LIN {X 0,Y 523.9,Z 252.85,A -85,B 0,C 180,E1 -4806.401,E2 -4806.401} C_VEL
LIN {X 0,Y 523.917,Z 252.846,A -85,B 0,C 180,E1 -4809.084,E2 -4809.084} C_VEL
LIN {X 0,Y 523.952,Z 252.837,A -85,B 0,C 180,E1 -4812.118,E2 -4812.118} C_VEL
LIN {X 0,Y 523.95,Z 252.839,A -85,B 0,C 180,E1 -4815.308,E2 -4815.308} C_VEL
LIN {X 0,Y 523.956,Z 252.84,A -85,B 0,C 180,E1 -4818.688,E2 -4818.688} C_VEL
LIN {X 0,Y 523.912,Z 252.849,A -85,B 0,C 180,E1 -4821.898,E2 -4821.898} C_VEL
LIN {X 0,Y 523.933,Z 252.83,A -85,B 0,C 180,E1 -4824.908,E2 -4824.908} C_VEL
LIN {X 0,Y 523.936,Z 252.838,A -85,B 0,C 180,E1 -4827.678,E2 -4827.678} C_VEL
LIN {X 0,Y 523.963,Z 252.839,A -85,B 0,C 180,E1 -4830.673,E2 -4830.673} C_VEL
LIN {X 0,Y 523.971,Z 252.84,A -85,B 0,C 180,E1 -4833.728,E2 -4833.728} C_VEL
LIN {X 0,Y 523.929,Z 252.844,A -85,B 0,C 180,E1 -4836.27,E2 -4836.27} C_VEL
LIN {X 0,Y 523.938,Z 252.84,A -85,B 0,C 180,E1 -4838.766,E2 -4838.766} C_VEL
LIN {X 0,Y 523.946,Z 252.842,A -85,B 0,C 180,E1 -4841.221,E2 -4841.221} C_VEL
LIN {X 0,Y 523.933,Z 252.845,A -85,B 0,C 180,E1 -4843.639,E2 -4843.639} C_VEL
LIN {X 0,Y 523.933,Z 252.847,A -85,B 0,C 180,E1 -4846.028,E2 -4846.028} C_VEL
LIN {X 0,Y 524.003,Z 252.831,A -85,B 0,C 180,E1 -4848.394,E2 -4848.394} C_VEL
LIN {X 0,Y 523.997,Z 252.838,A -85,B 0,C 180,E1 -4851.516,E2 -4851.516} C_VEL
LIN {X 0,Y 524.076,Z 252.822,A -85,B 0,C 180,E1 -4854.614,E2 -4854.614} C_VEL
LIN {X 0,Y 524.103,Z 252.827,A -85,B 0,C 180,E1 -4857.694,E2 -4857.694} C_VEL
LIN {X 0,Y 524.117,Z 252.819,A -85,B 0,C 180,E1 -4860.768,E2 -4860.768} C_VEL
LIN {X 0,Y 524.067,Z 252.823,A -85,B 0,C 180,E1 -4863.075,E2 -4863.075} C_VEL
LIN {X 0,Y 524.038,Z 252.829,A -85,B 0,C 180,E1 -4866.159,E2 -4866.159} C_VEL
LIN {X 0,Y 523.993,Z 252.837,A -85,B 0,C 180,E1 -4869.262,E2 -4869.262} C_VEL
LIN {X 0,Y 523.994,Z 252.837,A -85,B 0,C 180,E1 -4871.74,E2 -4871.74} C_VEL
LIN {X 0,Y 523.984,Z 252.838,A -85,B 0,C 180,E1 -4875.053,E2 -4875.053} C_VEL
LIN {X 0,Y 523.957,Z 252.839,A -85,B 0,C 180,E1 -4877.969,E2 -4877.969} C_VEL
LIN {X 0,Y 523.964,Z 252.836,A -85,B 0,C 180,E1 -4880.41,E2 -4880.41} C_VEL
LIN {X 0,Y 523.909,Z 252.849,A -85,B 0,C 180,E1 -4882.894,E2 -4882.894} C_VEL
LIN {X 0,Y 523.946,Z 252.84,A -85,B 0,C 180,E1 -4885.419,E2 -4885.419} C_VEL
LIN {X 0,Y 523.964,Z 252.838,A -85,B 0,C 180,E1 -4887.999,E2 -4887.999} C_VEL
LIN {X 0,Y 523.947,Z 252.845,A -85,B 0,C 180,E1 -4890.857,E2 -4890.857} C_VEL
LIN {X 0,Y 523.956,Z 252.827,A -85,B 0,C 180,E1 -4893.736,E2 -4893.736} C_VEL
LIN {X 0,Y 523.917,Z 252.844,A -85,B 0,C 180,E1 -4896.405,E2 -4896.405} C_VEL
LIN {X 0,Y 523.919,Z 252.845,A -85,B 0,C 180,E1 -4899.085,E2 -4899.085} C_VEL
LIN {X 0,Y 523.952,Z 252.831,A -85,B 0,C 180,E1 -4902.119,E2 -4902.119} C_VEL
LIN {X 0,Y 523.952,Z 252.841,A -85,B 0,C 180,E1 -4905.309,E2 -4905.309} C_VEL
LIN {X 0,Y 523.92,Z 252.841,A -85,B 0,C 180,E1 -4906.92,E2 -4906.92} C_VEL
LIN {X 0,Y 523.253,Z 252.921,A -85,B 0,C 180,E1 -4907.561,E2 -4907.561} C_VEL
LIN {X 0,Y 520.408,Z 253.282,A -85,B 0,C 180,E1 -4908.603,E2 -4908.603} C_VEL
LIN {X 0,Y 518.002,Z 253.587,A -85,B 0,C 180,E1 -4909.442,E2 -4909.442} C_VEL
LIN {X 0,Y 516.965,Z 253.716,A -85,B 0,C 180,E1 -4910.089,E2 -4910.089} C_VEL
LIN {X 0,Y 516.879,Z 253.725,A -85,B 0,C 180,E1 -4910.309,E2 -4910.309} C_VEL
LIN {X 0,Y 516.882,Z 253.721,A -85,B 0,C 180,E1 -4913.343,E2 -4913.343} C_VEL
LIN {X 0,Y 516.91,Z 253.719,A -85,B 0,C 180,E1 -4916.122,E2 -4916.122} C_VEL
LIN {X 0,Y 516.891,Z 253.723,A -85,B 0,C 180,E1 -4918.936,E2 -4918.936} C_VEL
LIN {X 0,Y 516.919,Z 253.712,A -85,B 0,C 180,E1 -4921.585,E2 -4921.585} C_VEL
LIN {X 0,Y 516.93,Z 253.717,A -85,B 0,C 180,E1 -4924.211,E2 -4924.211} C_VEL
LIN {X 0,Y 516.93,Z 253.837,A -85,B 0,C 180,E1 -4925.929,E2 -4925.929} C_VEL
LIN {X 0,Y 518.632,Z 262.689,A -85,B 0,C 180,E1 -4927.53,E2 -4927.53} C_VEL
LIN {X 0,Y 518.198,Z 277.695,A -85,B 0,C 180,E1 -4929.974,E2 -4929.974} C_VEL
LIN {X 0,Y 517.98,Z 286.774,A -85,B 0,C 180,E1 -4931.404,E2 -4931.404} C_VEL
LIN {X 0,Y 520.284,Z 298.799,A -85,B 0,C 180,E1 -4931.688,E2 -4931.688} C_VEL
LIN {X 0,Y 520.017,Z 379.819,A -85,B 0,C 180,E1 -4932.83,E2 -4932.83} C_VEL
LIN {X 0,Y 519.682,Z 424.477,A -85,B 0,C 180,E1 -4933.476,E2 -4933.476} C_VEL
LIN {X 0,Y 519.367,Z 439.105,A -85,B 0,C 180,E1 -4933.852,E2 -4933.852} C_VEL
LIN {X 0,Y 519.086,Z 453.266,A -85,B 0,C 180,E1 -4934.39,E2 -4934.39} C_VEL
LIN {X 0,Y 518.692,Z 466.922,A -85,B 0,C 180,E1 -4935.082,E2 -4935.082} C_VEL
LIN {X 0,Y 518.257,Z 479.18,A -85,B 0,C 180,E1 -4935.872,E2 -4935.872} C_VEL
LIN {X 0,Y 517.892,Z 490.403,A -85,B 0,C 180,E1 -4936.762,E2 -4936.762} C_VEL
LIN {X 0,Y 517.497,Z 501.263,A -85,B 0,C 180,E1 -4937.803,E2 -4937.803} C_VEL
LIN {X 0,Y 517.151,Z 511.76,A -85,B 0,C 180,E1 -4939.032,E2 -4939.032} C_VEL
LIN {X 0,Y 516.844,Z 520.123,A -85,B 0,C 180,E1 -4940.214,E2 -4940.214} C_VEL
LIN {X 0,Y 516.605,Z 528.11,A -85,B 0,C 180,E1 -4941.591,E2 -4941.591} C_VEL
LIN {X 0,Y 516.418,Z 534.54,A -85,B 0,C 180,E1 -4942.965,E2 -4942.965} C_VEL
LIN {X 0,Y 516.391,Z 540.243,A -85,B 0,C 180,E1 -4944.533,E2 -4944.533} C_VEL
LIN {X 0,Y 516.343,Z 544.391,A -85,B 0,C 180,E1 -4946.098,E2 -4946.098} C_VEL
LIN {X 0,Y 516.26,Z 547.108,A -85,B 0,C 180,E1 -4947.659,E2 -4947.659} C_VEL
LIN {X 0,Y 516.156,Z 548.474,A -85,B 0,C 180,E1 -4949.22,E2 -4949.22} C_VEL
LIN {X 0,Y 516.157,Z 548.517,A -85,B 0,C 180,E1 -4950.78,E2 -4950.78} C_VEL
LIN {X 0,Y 516.26,Z 547.233,A -85,B 0,C 180,E1 -4952.341,E2 -4952.341} C_VEL
LIN {X 0,Y 516.343,Z 544.592,A -85,B 0,C 180,E1 -4953.902,E2 -4953.902} C_VEL
LIN {X 0,Y 516.39,Z 540.527,A -85,B 0,C 180,E1 -4955.467,E2 -4955.467} C_VEL
LIN {X 0,Y 516.414,Z 534.911,A -85,B 0,C 180,E1 -4957.035,E2 -4957.035} C_VEL
LIN {X 0,Y 516.6,Z 528.569,A -85,B 0,C 180,E1 -4958.409,E2 -4958.409} C_VEL
LIN {X 0,Y 516.824,Z 520.683,A -85,B 0,C 180,E1 -4959.786,E2 -4959.786} C_VEL
LIN {X 0,Y 517.115,Z 512.434,A -85,B 0,C 180,E1 -4960.968,E2 -4960.968} C_VEL
LIN {X 0,Y 517.445,Z 502.412,A -85,B 0,C 180,E1 -4962.162,E2 -4962.162} C_VEL
LIN {X 0,Y 517.814,Z 491.436,A -85,B 0,C 180,E1 -4963.24,E2 -4963.24} C_VEL
LIN {X 0,Y 518.21,Z 480.425,A -85,B 0,C 180,E1 -4964.129,E2 -4964.129} C_VEL
LIN {X 0,Y 518.681,Z 468.481,A -85,B 0,C 180,E1 -4964.918,E2 -4964.918} C_VEL
LIN {X 0,Y 519.054,Z 455.296,A -85,B 0,C 180,E1 -4965.611,E2 -4965.611} C_VEL
LIN {X 0,Y 519.377,Z 441.413,A -85,B 0,C 180,E1 -4966.161,E2 -4966.161} C_VEL
LIN {X 0,Y 519.651,Z 427.406,A -85,B 0,C 180,E1 -4966.55,E2 -4966.55} C_VEL
LIN {X 0,Y 519.811,Z 409.431,A -85,B 0,C 180,E1 -4966.848,E2 -4966.848} C_VEL
LIN {X 0,Y 520.381,Z 299.087,A -85,B 0,C 180,E1 -4968.394,E2 -4968.394} C_VEL
LIN {X 0,Y 517.983,Z 286.806,A -85,B 0,C 180,E1 -4968.684,E2 -4968.684} C_VEL
LIN {X 0,Y 518.506,Z 269.351,A -85,B 0,C 180,E1 -4971.467,E2 -4971.467} C_VEL
LIN {X 0,Y 518.596,Z 262.055,A -85,B 0,C 180,E1 -4972.667,E2 -4972.667} C_VEL
LIN {X 0,Y 516.909,Z 253.814,A -85,B 0,C 180,E1 -4974.173,E2 -4974.173} C_VEL
LIN {X 0,Y 516.927,Z 253.719,A -85,B 0,C 180,E1 -4976.657,E2 -4976.657} C_VEL
LIN {X 0,Y 516.91,Z 253.719,A -85,B 0,C 180,E1 -4979.523,E2 -4979.523} C_VEL
LIN {X 0,Y 516.896,Z 253.72,A -85,B 0,C 180,E1 -4982.543,E2 -4982.543} C_VEL
LIN {X 0,Y 516.878,Z 253.725,A -85,B 0,C 180,E1 -4985.331,E2 -4985.331} C_VEL
LIN {X 0,Y 516.878,Z 253.722,A -85,B 0,C 180,E1 -4987.942,E2 -4987.942} C_VEL
LIN {X 0,Y 516.883,Z 253.722,A -85,B 0,C 180,E1 -4990.741,E2 -4990.741} C_VEL
LIN {X 0,Y 516.901,Z 253.712,A -85,B 0,C 180,E1 -4992.828,E2 -4992.828} C_VEL
LIN {X 0,Y 516.919,Z 253.719,A -85,B 0,C 180,E1 -4995.009,E2 -4995.009} C_VEL
LIN {X 0,Y 516.917,Z 253.706,A -85,B 0,C 180,E1 -4998.397,E2 -4998.397} C_VEL
LIN {X 0,Y 516.881,Z 253.727,A -85,B 0,C 180,E1 -5001.284,E2 -5001.284} C_VEL
LIN {X 0,Y 516.885,Z 253.718,A -85,B 0,C 180,E1 -5004.221,E2 -5004.221} C_VEL
LIN {X 0,Y 516.891,Z 253.711,A -85,B 0,C 180,E1 -5007.053,E2 -5007.053} C_VEL
LIN {X 0,Y 516.895,Z 253.719,A -85,B 0,C 180,E1 -5009.796,E2 -5009.796} C_VEL
LIN {X 0,Y 516.921,Z 253.717,A -85,B 0,C 180,E1 -5012.467,E2 -5012.467} C_VEL
LIN {X 0,Y 516.903,Z 253.724,A -85,B 0,C 180,E1 -5015.071,E2 -5015.071} C_VEL
LIN {X 0,Y 516.861,Z 253.723,A -85,B 0,C 180,E1 -5017.621,E2 -5017.621} C_VEL
LIN {X 0,Y 516.924,Z 253.712,A -85,B 0,C 180,E1 -5020.129,E2 -5020.129} C_VEL
LIN {X 0,Y 516.923,Z 253.72,A -85,B 0,C 180,E1 -5022.596,E2 -5022.596} C_VEL
LIN {X 0,Y 516.933,Z 253.716,A -85,B 0,C 180,E1 -5025.03,E2 -5025.03} C_VEL
LIN {X 0,Y 516.956,Z 253.713,A -85,B 0,C 180,E1 -5028.233,E2 -5028.233} C_VEL
LIN {X 0,Y 516.961,Z 253.706,A -85,B 0,C 180,E1 -5031.399,E2 -5031.399} C_VEL
LIN {X 0,Y 517.002,Z 253.705,A -85,B 0,C 180,E1 -5033.757,E2 -5033.757} C_VEL
LIN {X 0,Y 517.008,Z 253.703,A -85,B 0,C 180,E1 -5036.883,E2 -5036.883} C_VEL
LIN {X 0,Y 517.075,Z 253.697,A -85,B 0,C 180,E1 -5040,E2 -5040} C_VEL
LIN {X 0,Y 517.008,Z 253.701,A -85,B 0,C 180,E1 -5043.117,E2 -5043.117} C_VEL
LIN {X 0,Y 517.001,Z 253.71,A -85,B 0,C 180,E1 -5046.243,E2 -5046.243} C_VEL
LIN {X 0,Y 516.948,Z 253.709,A -85,B 0,C 180,E1 -5049.389,E2 -5049.389} C_VEL
LIN {X 0,Y 516.942,Z 253.712,A -85,B 0,C 180,E1 -5051.807,E2 -5051.807} C_VEL
LIN {X 0,Y 516.935,Z 253.712,A -85,B 0,C 180,E1 -5055.147,E2 -5055.147} C_VEL
LIN {X 0,Y 516.917,Z 253.723,A -85,B 0,C 180,E1 -5058.222,E2 -5058.222} C_VEL
LIN {X 0,Y 516.903,Z 253.717,A -85,B 0,C 180,E1 -5060.702,E2 -5060.702} C_VEL
LIN {X 0,Y 516.903,Z 253.725,A -85,B 0,C 180,E1 -5064.072,E2 -5064.072} C_VEL
LIN {X 0,Y 516.918,Z 253.714,A -85,B 0,C 180,E1 -5066.658,E2 -5066.658} C_VEL
LIN {X 0,Y 516.917,Z 253.718,A -85,B 0,C 180,E1 -5069.527,E2 -5069.527} C_VEL
LIN {X 0,Y 516.893,Z 253.713,A -85,B 0,C 180,E1 -5072.545,E2 -5072.545} C_VEL
LIN {X 0,Y 516.876,Z 253.71,A -85,B 0,C 180,E1 -5075.333,E2 -5075.333} C_VEL
LIN {X 0,Y 516.876,Z 253.729,A -85,B 0,C 180,E1 -5077.944,E2 -5077.944} C_VEL
LIN {X 0,Y 516.88,Z 253.718,A -85,B 0,C 180,E1 -5080.742,E2 -5080.742} C_VEL
LIN {X 0,Y 516.878,Z 253.721,A -85,B 0,C 180,E1 -5082.832,E2 -5082.832} C_VEL
LIN {X 0,Y 516.918,Z 253.716,A -85,B 0,C 180,E1 -5085.011,E2 -5085.011} C_VEL
LIN {X 0,Y 516.919,Z 253.71,A -85,B 0,C 180,E1 -5088.398,E2 -5088.398} C_VEL
LIN {X 0,Y 516.882,Z 253.726,A -85,B 0,C 180,E1 -5091.285,E2 -5091.285} C_VEL
LIN {X 0,Y 516.868,Z 253.724,A -85,B 0,C 180,E1 -5094.22,E2 -5094.22} C_VEL
LIN {X 0,Y 516.894,Z 253.719,A -85,B 0,C 180,E1 -5097.054,E2 -5097.054} C_VEL
LIN {X 0,Y 516.891,Z 253.709,A -85,B 0,C 180,E1 -5099.797,E2 -5099.797} C_VEL
LIN {X 0,Y 516.927,Z 253.719,A -85,B 0,C 180,E1 -5102.468,E2 -5102.468} C_VEL
LIN {X 0,Y 516.955,Z 253.758,A -85,B 0,C 180,E1 -5104.752,E2 -5104.752} C_VEL
LIN {X 0,Y 517.3,Z 255.393,A -85,B 0,C 180,E1 -5105.093,E2 -5105.093} C_VEL
LIN {X 0,Y 518.896,Z 263.487,A -85,B 0,C 180,E1 -5106.45,E2 -5106.45} C_VEL
LIN {X 0,Y 518.406,Z 279.65,A -85,B 0,C 180,E1 -5108.946,E2 -5108.946} C_VEL
LIN {X 0,Y 518.002,Z 295.678,A -85,B 0,C 180,E1 -5111.358,E2 -5111.358} C_VEL
LIN {X 0,Y 520.437,Z 309.426,A -85,B 0,C 180,E1 -5111.668,E2 -5111.668} C_VEL
LIN {X 0,Y 519.66,Z 433.577,A -85,B 0,C 180,E1 -5113.425,E2 -5113.425} C_VEL
LIN {X 0,Y 519.376,Z 447.528,A -85,B 0,C 180,E1 -5113.777,E2 -5113.777} C_VEL
LIN {X 0,Y 519.085,Z 461.402,A -85,B 0,C 180,E1 -5114.289,E2 -5114.289} C_VEL
LIN {X 0,Y 518.753,Z 473.578,A -85,B 0,C 180,E1 -5114.883,E2 -5114.883} C_VEL
LIN {X 0,Y 518.282,Z 486.388,A -85,B 0,C 180,E1 -5115.672,E2 -5115.672} C_VEL
LIN {X 0,Y 517.89,Z 498.036,A -85,B 0,C 180,E1 -5116.562,E2 -5116.562} C_VEL
LIN {X 0,Y 517.493,Z 508.974,A -85,B 0,C 180,E1 -5117.577,E2 -5117.577} C_VEL
LIN {X 0,Y 517.235,Z 518.468,A -85,B 0,C 180,E1 -5118.638,E2 -5118.638} C_VEL
LIN {X 0,Y 516.849,Z 527.332,A -85,B 0,C 180,E1 -5119.819,E2 -5119.819} C_VEL
LIN {X 0,Y 516.683,Z 534.708,A -85,B 0,C 180,E1 -5121.001,E2 -5121.001} C_VEL
LIN {X 0,Y 516.495,Z 540.857,A -85,B 0,C 180,E1 -5122.18,E2 -5122.18} C_VEL
LIN {X 0,Y 516.382,Z 547.387,A -85,B 0,C 180,E1 -5123.749,E2 -5123.749} C_VEL
LIN {X 0,Y 516.305,Z 551.207,A -85,B 0,C 180,E1 -5124.924,E2 -5124.924} C_VEL
LIN {X 0,Y 516.324,Z 554.15,A -85,B 0,C 180,E1 -5126.098,E2 -5126.098} C_VEL
LIN {X 0,Y 516.259,Z 556.844,A -85,B 0,C 180,E1 -5127.659,E2 -5127.659} C_VEL
LIN {X 0,Y 516.157,Z 558.178,A -85,B 0,C 180,E1 -5129.22,E2 -5129.22} C_VEL
LIN {X 0,Y 516.157,Z 558.178,A -85,B 0,C 180,E1 -5130.78,E2 -5130.78} C_VEL
LIN {X 0,Y 516.26,Z 556.847,A -85,B 0,C 180,E1 -5132.341,E2 -5132.341} C_VEL
LIN {X 0,Y 516.324,Z 554.154,A -85,B 0,C 180,E1 -5133.902,E2 -5133.902} C_VEL
LIN {X 0,Y 516.382,Z 550.026,A -85,B 0,C 180,E1 -5135.467,E2 -5135.467} C_VEL
LIN {X 0,Y 516.402,Z 544.337,A -85,B 0,C 180,E1 -5137.035,E2 -5137.035} C_VEL
LIN {X 0,Y 516.582,Z 537.923,A -85,B 0,C 180,E1 -5138.41,E2 -5138.41} C_VEL
LIN {X 0,Y 516.805,Z 529.954,A -85,B 0,C 180,E1 -5139.787,E2 -5139.787} C_VEL
LIN {X 0,Y 517.101,Z 521.618,A -85,B 0,C 180,E1 -5140.969,E2 -5140.969} C_VEL
LIN {X 0,Y 517.456,Z 511.182,A -85,B 0,C 180,E1 -5142.197,E2 -5142.197} C_VEL
LIN {X 0,Y 517.824,Z 500.382,A -85,B 0,C 180,E1 -5143.24,E2 -5143.24} C_VEL
LIN {X 0,Y 518.245,Z 487.817,A -85,B 0,C 180,E1 -5144.229,E2 -5144.229} C_VEL
LIN {X 0,Y 518.7,Z 475.343,A -85,B 0,C 180,E1 -5145.018,E2 -5145.018} C_VEL
LIN {X 0,Y 519.077,Z 462.519,A -85,B 0,C 180,E1 -5145.661,E2 -5145.661} C_VEL
LIN {X 0,Y 519.367,Z 448.602,A -85,B 0,C 180,E1 -5146.188,E2 -5146.188} C_VEL
LIN {X 0,Y 519.65,Z 434.709,A -85,B 0,C 180,E1 -5146.55,E2 -5146.55} C_VEL
LIN {X 0,Y 519.847,Z 408.415,A -85,B 0,C 180,E1 -5146.948,E2 -5146.948} C_VEL
LIN {X 0,Y 520.279,Z 308.185,A -85,B 0,C 180,E1 -5148.355,E2 -5148.355} C_VEL
LIN {X 0,Y 517.994,Z 295.748,A -85,B 0,C 180,E1 -5148.638,E2 -5148.638} C_VEL
LIN {X 0,Y 518.507,Z 276.952,A -85,B 0,C 180,E1 -5151.467,E2 -5151.467} C_VEL
LIN {X 0,Y 518.89,Z 263.487,A -85,B 0,C 180,E1 -5153.55,E2 -5153.55} C_VEL
LIN {X 0,Y 517.034,Z 254.105,A -85,B 0,C 180,E1 -5155.136,E2 -5155.136} C_VEL
LIN {X 0,Y 516.954,Z 253.708,A -85,B 0,C 180,E1 -5155.356,E2 -5155.356} C_VEL
LIN {X 0,Y 516.918,Z 253.718,A -85,B 0,C 180,E1 -5158.415,E2 -5158.415} C_VEL
LIN {X 0,Y 516.888,Z 253.723,A -85,B 0,C 180,E1 -5161.109,E2 -5161.109} C_VEL
LIN {X 0,Y 516.906,Z 253.716,A -85,B 0,C 180,E1 -5163.966,E2 -5163.966} C_VEL
LIN {X 0,Y 516.873,Z 253.722,A -85,B 0,C 180,E1 -5166.745,E2 -5166.745} C_VEL
LIN {X 0,Y 516.878,Z 253.722,A -85,B 0,C 180,E1 -5169.721,E2 -5169.721} C_VEL
LIN {X 0,Y 516.902,Z 253.721,A -85,B 0,C 180,E1 -5172.76,E2 -5172.76} C_VEL
LIN {X 0,Y 516.918,Z 253.716,A -85,B 0,C 180,E1 -5175.009,E2 -5175.009} C_VEL
LIN {X 0,Y 516.912,Z 253.721,A -85,B 0,C 180,E1 -5178.398,E2 -5178.398} C_VEL
LIN {X 0,Y 516.878,Z 253.721,A -85,B 0,C 180,E1 -5181.284,E2 -5181.284} C_VEL
LIN {X 0,Y 516.885,Z 253.715,A -85,B 0,C 180,E1 -5184.221,E2 -5184.221} C_VEL
LIN {X 0,Y 516.891,Z 253.712,A -85,B 0,C 180,E1 -5187.053,E2 -5187.053} C_VEL
LIN {X 0,Y 516.895,Z 253.723,A -85,B 0,C 180,E1 -5189.797,E2 -5189.797} C_VEL
LIN {X 0,Y 516.923,Z 253.715,A -85,B 0,C 180,E1 -5192.467,E2 -5192.467} C_VEL
LIN {X 0,Y 516.904,Z 253.718,A -85,B 0,C 180,E1 -5195.072,E2 -5195.072} C_VEL
LIN {X 0,Y 516.878,Z 253.721,A -85,B 0,C 180,E1 -5198.462,E2 -5198.462} C_VEL
LIN {X 0,Y 516.897,Z 253.719,A -85,B 0,C 180,E1 -5200.955,E2 -5200.955} C_VEL
LIN {X 0,Y 516.909,Z 253.717,A -85,B 0,C 180,E1 -5203.41,E2 -5203.41} C_VEL
LIN {X 0,Y 516.888,Z 253.728,A -85,B 0,C 180,E1 -5205.833,E2 -5205.833} C_VEL
LIN {X 0,Y 516.957,Z 253.71,A -85,B 0,C 180,E1 -5208.234,E2 -5208.234} C_VEL
LIN {X 0,Y 516.962,Z 253.712,A -85,B 0,C 180,E1 -5211.4,E2 -5211.4} C_VEL
LIN {X 0,Y 517.002,Z 253.71,A -85,B 0,C 180,E1 -5213.757,E2 -5213.757} C_VEL
LIN {X 0,Y 517.076,Z 253.703,A -85,B 0,C 180,E1 -5217.663,E2 -5217.663} C_VEL
LIN {X 0,Y 517.087,Z 253.694,A -85,B 0,C 180,E1 -5220.779,E2 -5220.779} C_VEL
LIN {X 0,Y 517.008,Z 253.702,A -85,B 0,C 180,E1 -5223.117,E2 -5223.117} C_VEL
LIN {X 0,Y 517.002,Z 253.705,A -85,B 0,C 180,E1 -5226.243,E2 -5226.243} C_VEL
LIN {X 0,Y 516.947,Z 253.715,A -85,B 0,C 180,E1 -5229.389,E2 -5229.389} C_VEL
LIN {X 0,Y 516.944,Z 253.715,A -85,B 0,C 180,E1 -5231.808,E2 -5231.808} C_VEL
LIN {X 0,Y 516.936,Z 253.716,A -85,B 0,C 180,E1 -5235.147,E2 -5235.147} C_VEL
LIN {X 0,Y 516.918,Z 253.716,A -85,B 0,C 180,E1 -5238.223,E2 -5238.223} C_VEL
LIN {X 0,Y 516.905,Z 253.717,A -85,B 0,C 180,E1 -5240.702,E2 -5240.702} C_VEL
LIN {X 0,Y 516.904,Z 253.718,A -85,B 0,C 180,E1 -5244.072,E2 -5244.072} C_VEL
LIN {X 0,Y 516.92,Z 253.715,A -85,B 0,C 180,E1 -5246.658,E2 -5246.658} C_VEL
LIN {X 0,Y 516.919,Z 253.717,A -85,B 0,C 180,E1 -5249.527,E2 -5249.527} C_VEL
LIN {X 0,Y 516.895,Z 253.715,A -85,B 0,C 180,E1 -5252.545,E2 -5252.545} C_VEL
LIN {X 0,Y 516.878,Z 253.72,A -85,B 0,C 180,E1 -5255.333,E2 -5255.333} C_VEL
LIN {X 0,Y 516.877,Z 253.722,A -85,B 0,C 180,E1 -5257.944,E2 -5257.944} C_VEL
LIN {X 0,Y 516.899,Z 253.715,A -85,B 0,C 180,E1 -5260.74,E2 -5260.74} C_VEL
LIN {X 0,Y 516.879,Z 253.72,A -85,B 0,C 180,E1 -5263.904,E2 -5263.904} C_VEL
LIN {X 0,Y 516.879,Z 253.722,A -85,B 0,C 180,E1 -5266.108,E2 -5266.108} C_VEL
LIN {X 0,Y 516.915,Z 253.714,A -85,B 0,C 180,E1 -5268.399,E2 -5268.399} C_VEL
LIN {X 0,Y 516.879,Z 253.725,A -85,B 0,C 180,E1 -5270.309,E2 -5270.309} C_VEL
LIN {X 0,Y 516.209,Z 253.807,A -85,B 0,C 180,E1 -5270.959,E2 -5270.959} C_VEL
LIN {X 0,Y 513.364,Z 254.159,A -85,B 0,C 180,E1 -5272.015,E2 -5272.015} C_VEL
LIN {X 0,Y 510.956,Z 254.463,A -85,B 0,C 180,E1 -5272.865,E2 -5272.865} C_VEL
LIN {X 0,Y 509.916,Z 254.589,A -85,B 0,C 180,E1 -5273.521,E2 -5273.521} C_VEL
LIN {X 0,Y 509.828,Z 254.6,A -85,B 0,C 180,E1 -5273.744,E2 -5273.744} C_VEL
LIN {X 0,Y 509.86,Z 254.6,A -85,B 0,C 180,E1 -5276.54,E2 -5276.54} C_VEL
LIN {X 0,Y 509.845,Z 254.599,A -85,B 0,C 180,E1 -5279.335,E2 -5279.335} C_VEL
LIN {X 0,Y 509.894,Z 254.585,A -85,B 0,C 180,E1 -5282.055,E2 -5282.055} C_VEL
LIN {X 0,Y 509.841,Z 254.593,A -85,B 0,C 180,E1 -5284.703,E2 -5284.703} C_VEL
LIN {X 0,Y 509.875,Z 254.64,A -85,B 0,C 180,E1 -5285.683,E2 -5285.683} C_VEL
LIN {X 0,Y 510.429,Z 257.459,A -85,B 0,C 180,E1 -5286.251,E2 -5286.251} C_VEL
LIN {X 0,Y 511.783,Z 265.056,A -85,B 0,C 180,E1 -5287.6,E2 -5287.6} C_VEL
LIN {X 0,Y 511.126,Z 282.841,A -85,B 0,C 180,E1 -5290.523,E2 -5290.523} C_VEL
LIN {X 0,Y 511.067,Z 286.884,A -85,B 0,C 180,E1 -5291.146,E2 -5291.146} C_VEL
LIN {X 0,Y 513.675,Z 300.421,A -85,B 0,C 180,E1 -5291.466,E2 -5291.466} C_VEL
LIN {X 0,Y 512.899,Z 423.387,A -85,B 0,C 180,E1 -5293.226,E2 -5293.226} C_VEL
LIN {X 0,Y 512.57,Z 438.113,A -85,B 0,C 180,E1 -5293.596,E2 -5293.596} C_VEL
LIN {X 0,Y 512.284,Z 452.218,A -85,B 0,C 180,E1 -5294.126,E2 -5294.126} C_VEL
LIN {X 0,Y 511.912,Z 465.234,A -85,B 0,C 180,E1 -5294.778,E2 -5294.778} C_VEL
LIN {X 0,Y 511.412,Z 477.832,A -85,B 0,C 180,E1 -5295.577,E2 -5295.577} C_VEL
LIN {X 0,Y 510.999,Z 489.305,A -85,B 0,C 180,E1 -5296.479,E2 -5296.479} C_VEL
LIN {X 0,Y 510.55,Z 499.789,A -85,B 0,C 180,E1 -5297.474,E2 -5297.474} C_VEL
LIN {X 0,Y 510.208,Z 510.284,A -85,B 0,C 180,E1 -5298.68,E2 -5298.68} C_VEL
LIN {X 0,Y 509.836,Z 518.905,A -85,B 0,C 180,E1 -5299.878,E2 -5299.878} C_VEL
LIN {X 0,Y 509.602,Z 527.17,A -85,B 0,C 180,E1 -5301.275,E2 -5301.275} C_VEL
LIN {X 0,Y 509.413,Z 532.927,A -85,B 0,C 180,E1 -5302.469,E2 -5302.469} C_VEL
LIN {X 0,Y 509.308,Z 537.665,A -85,B 0,C 180,E1 -5303.662,E2 -5303.662} C_VEL
LIN {X 0,Y 509.239,Z 541.51,A -85,B 0,C 180,E1 -5304.853,E2 -5304.853} C_VEL
LIN {X 0,Y 509.251,Z 544.459,A -85,B 0,C 180,E1 -5306.043,E2 -5306.043} C_VEL
LIN {X 0,Y 509.189,Z 547.175,A -85,B 0,C 180,E1 -5307.627,E2 -5307.627} C_VEL
LIN {X 0,Y 509.07,Z 548.541,A -85,B 0,C 180,E1 -5309.209,E2 -5309.209} C_VEL
LIN {X 0,Y 509.071,Z 548.584,A -85,B 0,C 180,E1 -5310.791,E2 -5310.791} C_VEL
LIN {X 0,Y 509.188,Z 547.299,A -85,B 0,C 180,E1 -5312.373,E2 -5312.373} C_VEL
LIN {X 0,Y 509.251,Z 544.657,A -85,B 0,C 180,E1 -5313.957,E2 -5313.957} C_VEL
LIN {X 0,Y 509.327,Z 540.592,A -85,B 0,C 180,E1 -5315.543,E2 -5315.543} C_VEL
LIN {X 0,Y 509.361,Z 534.975,A -85,B 0,C 180,E1 -5317.133,E2 -5317.133} C_VEL
LIN {X 0,Y 509.557,Z 528.633,A -85,B 0,C 180,E1 -5318.526,E2 -5318.526} C_VEL
LIN {X 0,Y 509.783,Z 520.746,A -85,B 0,C 180,E1 -5319.923,E2 -5319.923} C_VEL
LIN {X 0,Y 510.114,Z 512.496,A -85,B 0,C 180,E1 -5321.121,E2 -5321.121} C_VEL
LIN {X 0,Y 510.455,Z 502.828,A -85,B 0,C 180,E1 -5322.291,E2 -5322.291} C_VEL
LIN {X 0,Y 510.898,Z 491.496,A -85,B 0,C 180,E1 -5323.422,E2 -5323.422} C_VEL
LIN {X 0,Y 511.314,Z 480.484,A -85,B 0,C 180,E1 -5324.324,E2 -5324.324} C_VEL
LIN {X 0,Y 511.819,Z 468.537,A -85,B 0,C 180,E1 -5325.123,E2 -5325.123} C_VEL
LIN {X 0,Y 512.219,Z 455.348,A -85,B 0,C 180,E1 -5325.825,E2 -5325.825} C_VEL
LIN {X 0,Y 512.557,Z 441.104,A -85,B 0,C 180,E1 -5326.394,E2 -5326.394} C_VEL
LIN {X 0,Y 512.841,Z 427.444,A -85,B 0,C 180,E1 -5326.776,E2 -5326.776} C_VEL
LIN {X 0,Y 513.01,Z 407.664,A -85,B 0,C 180,E1 -5327.104,E2 -5327.104} C_VEL
LIN {X 0,Y 513.652,Z 299.991,A -85,B 0,C 180,E1 -5328.631,E2 -5328.631} C_VEL
LIN {X 0,Y 511.089,Z 287.082,A -85,B 0,C 180,E1 -5328.933,E2 -5328.933} C_VEL
LIN {X 0,Y 511.095,Z 284.659,A -85,B 0,C 180,E1 -5329.27,E2 -5329.27} C_VEL
LIN {X 0,Y 511.794,Z 265.599,A -85,B 0,C 180,E1 -5332.399,E2 -5332.399} C_VEL
LIN {X 0,Y 510.847,Z 259.261,A -85,B 0,C 180,E1 -5333.513,E2 -5333.513} C_VEL
LIN {X 0,Y 509.878,Z 254.731,A -85,B 0,C 180,E1 -5334.371,E2 -5334.371} C_VEL
LIN {X 0,Y 509.886,Z 254.596,A -85,B 0,C 180,E1 -5337.055,E2 -5337.055} C_VEL
LIN {X 0,Y 509.856,Z 254.602,A -85,B 0,C 180,E1 -5339.75,E2 -5339.75} C_VEL
LIN {X 0,Y 509.873,Z 254.595,A -85,B 0,C 180,E1 -5342.774,E2 -5342.774} C_VEL
LIN {X 0,Y 509.837,Z 254.606,A -85,B 0,C 180,E1 -5345.58,E2 -5345.58} C_VEL
LIN {X 0,Y 509.847,Z 254.595,A -85,B 0,C 180,E1 -5348.337,E2 -5348.337} C_VEL
LIN {X 0,Y 509.855,Z 254.598,A -85,B 0,C 180,E1 -5351.424,E2 -5351.424} C_VEL
LIN {X 0,Y 509.853,Z 254.596,A -85,B 0,C 180,E1 -5354.667,E2 -5354.667} C_VEL
LIN {X 0,Y 509.856,Z 254.585,A -85,B 0,C 180,E1 -5358.102,E2 -5358.102} C_VEL
LIN {X 0,Y 509.854,Z 254.594,A -85,B 0,C 180,E1 -5360.648,E2 -5360.648} C_VEL
LIN {X 0,Y 509.83,Z 254.6,A -85,B 0,C 180,E1 -5363.647,E2 -5363.647} C_VEL
LIN {X 0,Y 509.856,Z 254.584,A -85,B 0,C 180,E1 -5366.539,E2 -5366.539} C_VEL
LIN {X 0,Y 509.844,Z 254.603,A -85,B 0,C 180,E1 -5369.334,E2 -5369.334} C_VEL
LIN {X 0,Y 509.887,Z 254.592,A -85,B 0,C 180,E1 -5372.054,E2 -5372.054} C_VEL
LIN {X 0,Y 509.869,Z 254.594,A -85,B 0,C 180,E1 -5374.703,E2 -5374.703} C_VEL
LIN {X 0,Y 509.819,Z 254.601,A -85,B 0,C 180,E1 -5377.457,E2 -5377.457} C_VEL
LIN {X 0,Y 509.908,Z 254.586,A -85,B 0,C 180,E1 -5379.844,E2 -5379.844} C_VEL
LIN {X 0,Y 509.879,Z 254.595,A -85,B 0,C 180,E1 -5383.174,E2 -5383.174} C_VEL
LIN {X 0,Y 509.855,Z 254.592,A -85,B 0,C 180,E1 -5385.634,E2 -5385.634} C_VEL
LIN {X 0,Y 509.909,Z 254.594,A -85,B 0,C 180,E1 -5388.874,E2 -5388.874} C_VEL
LIN {X 0,Y 509.942,Z 254.581,A -85,B 0,C 180,E1 -5392.078,E2 -5392.078} C_VEL
LIN {X 0,Y 509.984,Z 254.586,A -85,B 0,C 180,E1 -5394.464,E2 -5394.464} C_VEL
LIN {X 0,Y 510.046,Z 254.565,A -85,B 0,C 180,E1 -5397.631,E2 -5397.631} C_VEL
LIN {X 0,Y 510.057,Z 254.575,A -85,B 0,C 180,E1 -5400.789,E2 -5400.789} C_VEL
LIN {X 0,Y 509.95,Z 254.58,A -85,B 0,C 180,E1 -5403.16,E2 -5403.16} C_VEL
LIN {X 0,Y 509.97,Z 254.587,A -85,B 0,C 180,E1 -5406.33,E2 -5406.33} C_VEL
LIN {X 0,Y 509.909,Z 254.589,A -85,B 0,C 180,E1 -5408.72,E2 -5408.72} C_VEL
LIN {X 0,Y 509.895,Z 254.591,A -85,B 0,C 180,E1 -5411.932,E2 -5411.932} C_VEL
LIN {X 0,Y 509.884,Z 254.59,A -85,B 0,C 180,E1 -5415.242,E2 -5415.242} C_VEL
LIN {X 0,Y 509.88,Z 254.595,A -85,B 0,C 180,E1 -5418.001,E2 -5418.001} C_VEL
LIN {X 0,Y 509.841,Z 254.595,A -85,B 0,C 180,E1 -5421.002,E2 -5421.002} C_VEL
LIN {X 0,Y 509.828,Z 254.599,A -85,B 0,C 180,E1 -5423.564,E2 -5423.564} C_VEL
LIN {X 0,Y 509.904,Z 254.59,A -85,B 0,C 180,E1 -5426.379,E2 -5426.379} C_VEL
LIN {X 0,Y 509.878,Z 254.593,A -85,B 0,C 180,E1 -5428.844,E2 -5428.844} C_VEL
LIN {X 0,Y 509.82,Z 254.603,A -85,B 0,C 180,E1 -5431.59,E2 -5431.59} C_VEL
LIN {X 0,Y 509.847,Z 254.585,A -85,B 0,C 180,E1 -5434.414,E2 -5434.414} C_VEL
LIN {X 0,Y 509.813,Z 254.601,A -85,B 0,C 180,E1 -5437.341,E2 -5437.341} C_VEL
LIN {X 0,Y 509.833,Z 254.598,A -85,B 0,C 180,E1 -5440.383,E2 -5440.383} C_VEL
LIN {X 0,Y 509.818,Z 254.602,A -85,B 0,C 180,E1 -5443.063,E2 -5443.063} C_VEL
LIN {X 0,Y 509.827,Z 254.606,A -85,B 0,C 180,E1 -5445.793,E2 -5445.793} C_VEL
LIN {X 0,Y 509.862,Z 254.588,A -85,B 0,C 180,E1 -5448.576,E2 -5448.576} C_VEL
LIN {X 0,Y 509.848,Z 254.598,A -85,B 0,C 180,E1 -5451.787,E2 -5451.787} C_VEL
LIN {X 0,Y 509.827,Z 254.601,A -85,B 0,C 180,E1 -5454.623,E2 -5454.623} C_VEL
LIN {X 0,Y 509.861,Z 254.602,A -85,B 0,C 180,E1 -5457.482,E2 -5457.482} C_VEL
LIN {X 0,Y 509.857,Z 254.582,A -85,B 0,C 180,E1 -5460.274,E2 -5460.274} C_VEL
LIN {X 0,Y 509.884,Z 254.593,A -85,B 0,C 180,E1 -5462.945,E2 -5462.945} C_VEL
LIN {X 0,Y 509.955,Z 254.811,A -85,B 0,C 180,E1 -5464.6,E2 -5464.6} C_VEL
LIN {X 0,Y 511.982,Z 264.774,A -85,B 0,C 180,E1 -5466.328,E2 -5466.328} C_VEL
LIN {X 0,Y 511.528,Z 279.589,A -85,B 0,C 180,E1 -5468.649,E2 -5468.649} C_VEL
LIN {X 0,Y 511.07,Z 295.584,A -85,B 0,C 180,E1 -5471.094,E2 -5471.094} C_VEL
LIN {X 0,Y 513.688,Z 310.506,A -85,B 0,C 180,E1 -5471.435,E2 -5471.435} C_VEL
LIN {X 0,Y 512.864,Z 433.51,A -85,B 0,C 180,E1 -5473.199,E2 -5473.199} C_VEL
LIN {X 0,Y 512.557,Z 447.779,A -85,B 0,C 180,E1 -5473.565,E2 -5473.565} C_VEL
LIN {X 0,Y 512.245,Z 461.335,A -85,B 0,C 180,E1 -5474.074,E2 -5474.074} C_VEL
LIN {X 0,Y 511.878,Z 473.511,A -85,B 0,C 180,E1 -5474.675,E2 -5474.675} C_VEL
LIN {X 0,Y 511.378,Z 486.322,A -85,B 0,C 180,E1 -5475.475,E2 -5475.475} C_VEL
LIN {X 0,Y 510.929,Z 497.969,A -85,B 0,C 180,E1 -5476.376,E2 -5476.376} C_VEL
LIN {X 0,Y 510.532,Z 508.712,A -85,B 0,C 180,E1 -5477.385,E2 -5477.385} C_VEL
LIN {X 0,Y 510.227,Z 518.401,A -85,B 0,C 180,E1 -5478.479,E2 -5478.479} C_VEL
LIN {X 0,Y 509.826,Z 527.265,A -85,B 0,C 180,E1 -5479.677,E2 -5479.677} C_VEL
LIN {X 0,Y 509.588,Z 535.759,A -85,B 0,C 180,E1 -5481.074,E2 -5481.074} C_VEL
LIN {X 0,Y 509.369,Z 542.603,A -85,B 0,C 180,E1 -5482.468,E2 -5482.468} C_VEL
LIN {X 0,Y 509.29,Z 548.715,A -85,B 0,C 180,E1 -5484.06,E2 -5484.06} C_VEL
LIN {X 0,Y 509.18,Z 552.206,A -85,B 0,C 180,E1 -5485.25,E2 -5485.25} C_VEL
LIN {X 0,Y 509.193,Z 555.603,A -85,B 0,C 180,E1 -5486.835,E2 -5486.835} C_VEL
LIN {X 0,Y 509.109,Z 557.612,A -85,B 0,C 180,E1 -5488.418,E2 -5488.418} C_VEL
LIN {X 0,Y 509.064,Z 558.278,A -85,B 0,C 180,E1 -5490,E2 -5490} C_VEL
LIN {X 0,Y 509.109,Z 557.614,A -85,B 0,C 180,E1 -5491.582,E2 -5491.582} C_VEL
LIN {X 0,Y 509.193,Z 555.607,A -85,B 0,C 180,E1 -5493.165,E2 -5493.165} C_VEL
LIN {X 0,Y 509.181,Z 552.209,A -85,B 0,C 180,E1 -5494.75,E2 -5494.75} C_VEL
LIN {X 0,Y 509.312,Z 548.714,A -85,B 0,C 180,E1 -5495.94,E2 -5495.94} C_VEL
LIN {X 0,Y 509.327,Z 544.27,A -85,B 0,C 180,E1 -5497.134,E2 -5497.134} C_VEL
LIN {X 0,Y 509.54,Z 537.857,A -85,B 0,C 180,E1 -5498.527,E2 -5498.527} C_VEL
LIN {X 0,Y 509.744,Z 529.887,A -85,B 0,C 180,E1 -5499.924,E2 -5499.924} C_VEL
LIN {X 0,Y 510.091,Z 521.551,A -85,B 0,C 180,E1 -5501.121,E2 -5501.121} C_VEL
LIN {X 0,Y 510.458,Z 511.463,A -85,B 0,C 180,E1 -5502.327,E2 -5502.327} C_VEL
LIN {X 0,Y 510.881,Z 500.316,A -85,B 0,C 180,E1 -5503.423,E2 -5503.423} C_VEL
LIN {X 0,Y 511.316,Z 487.75,A -85,B 0,C 180,E1 -5504.426,E2 -5504.426} C_VEL
LIN {X 0,Y 511.81,Z 475.276,A -85,B 0,C 180,E1 -5505.225,E2 -5505.225} C_VEL
LIN {X 0,Y 512.247,Z 462.453,A -85,B 0,C 180,E1 -5505.875,E2 -5505.875} C_VEL
LIN {X 0,Y 512.566,Z 448.397,A -85,B 0,C 180,E1 -5506.413,E2 -5506.413} C_VEL
LIN {X 0,Y 512.839,Z 434.643,A -85,B 0,C 180,E1 -5506.776,E2 -5506.776} C_VEL
LIN {X 0,Y 513.081,Z 408.349,A -85,B 0,C 180,E1 -5507.178,E2 -5507.178} C_VEL
LIN {X 0,Y 513.638,Z 309.663,A -85,B 0,C 180,E1 -5508.579,E2 -5508.579} C_VEL
LIN {X 0,Y 511.073,Z 295.599,A -85,B 0,C 180,E1 -5508.905,E2 -5508.905} C_VEL
LIN {X 0,Y 511.623,Z 276.892,A -85,B 0,C 180,E1 -5511.77,E2 -5511.77} C_VEL
LIN {X 0,Y 511.982,Z 264.773,A -85,B 0,C 180,E1 -5513.672,E2 -5513.672} C_VEL
LIN {X 0,Y 509.955,Z 254.811,A -85,B 0,C 180,E1 -5515.401,E2 -5515.401} C_VEL
LIN {X 0,Y 509.884,Z 254.593,A -85,B 0,C 180,E1 -5517.055,E2 -5517.055} C_VEL
LIN {X 0,Y 509.856,Z 254.582,A -85,B 0,C 180,E1 -5519.75,E2 -5519.75} C_VEL
LIN {X 0,Y 509.873,Z 254.596,A -85,B 0,C 180,E1 -5522.774,E2 -5522.774} C_VEL
LIN {X 0,Y 509.823,Z 254.601,A -85,B 0,C 180,E1 -5525.578,E2 -5525.578} C_VEL
LIN {X 0,Y 509.846,Z 254.601,A -85,B 0,C 180,E1 -5528.337,E2 -5528.337} C_VEL
LIN {X 0,Y 509.853,Z 254.588,A -85,B 0,C 180,E1 -5531.425,E2 -5531.425} C_VEL
LIN {X 0,Y 509.853,Z 254.6,A -85,B 0,C 180,E1 -5534.667,E2 -5534.667} C_VEL
LIN {X 0,Y 509.853,Z 254.603,A -85,B 0,C 180,E1 -5538.102,E2 -5538.102} C_VEL
LIN {X 0,Y 509.843,Z 254.601,A -85,B 0,C 180,E1 -5540.647,E2 -5540.647} C_VEL
LIN {X 0,Y 509.83,Z 254.598,A -85,B 0,C 180,E1 -5543.647,E2 -5543.647} C_VEL
LIN {X 0,Y 509.856,Z 254.592,A -85,B 0,C 180,E1 -5546.539,E2 -5546.539} C_VEL
LIN {X 0,Y 509.844,Z 254.597,A -85,B 0,C 180,E1 -5549.334,E2 -5549.334} C_VEL
LIN {X 0,Y 509.888,Z 254.595,A -85,B 0,C 180,E1 -5552.054,E2 -5552.054} C_VEL
LIN {X 0,Y 509.871,Z 254.595,A -85,B 0,C 180,E1 -5554.704,E2 -5554.704} C_VEL
LIN {X 0,Y 509.829,Z 254.599,A -85,B 0,C 180,E1 -5557.455,E2 -5557.455} C_VEL
LIN {X 0,Y 509.908,Z 254.596,A -85,B 0,C 180,E1 -5559.844,E2 -5559.844} C_VEL
LIN {X 0,Y 509.879,Z 254.59,A -85,B 0,C 180,E1 -5563.175,E2 -5563.175} C_VEL
LIN {X 0,Y 509.856,Z 254.6,A -85,B 0,C 180,E1 -5565.634,E2 -5565.634} C_VEL
LIN {X 0,Y 509.905,Z 254.586,A -85,B 0,C 180,E1 -5568.874,E2 -5568.874} C_VEL
LIN {X 0,Y 509.943,Z 254.588,A -85,B 0,C 180,E1 -5572.078,E2 -5572.078} C_VEL
LIN {X 0,Y 509.975,Z 254.578,A -85,B 0,C 180,E1 -5574.464,E2 -5574.464} C_VEL
LIN {X 0,Y 510.047,Z 254.578,A -85,B 0,C 180,E1 -5577.631,E2 -5577.631} C_VEL
LIN {X 0,Y 510.057,Z 254.57,A -85,B 0,C 180,E1 -5580.79,E2 -5580.79} C_VEL
LIN {X 0,Y 509.95,Z 254.581,A -85,B 0,C 180,E1 -5583.16,E2 -5583.16} C_VEL
LIN {X 0,Y 509.97,Z 254.581,A -85,B 0,C 180,E1 -5586.33,E2 -5586.33} C_VEL
LIN {X 0,Y 509.908,Z 254.585,A -85,B 0,C 180,E1 -5588.72,E2 -5588.72} C_VEL
LIN {X 0,Y 509.896,Z 254.592,A -85,B 0,C 180,E1 -5591.932,E2 -5591.932} C_VEL
LIN {X 0,Y 509.885,Z 254.594,A -85,B 0,C 180,E1 -5595.242,E2 -5595.242} C_VEL
LIN {X 0,Y 509.881,Z 254.593,A -85,B 0,C 180,E1 -5598.001,E2 -5598.001} C_VEL
LIN {X 0,Y 509.843,Z 254.599,A -85,B 0,C 180,E1 -5601.002,E2 -5601.002} C_VEL
LIN {X 0,Y 509.862,Z 254.596,A -85,B 0,C 180,E1 -5604.426,E2 -5604.426} C_VEL
LIN {X 0,Y 509.879,Z 254.597,A -85,B 0,C 180,E1 -5607.056,E2 -5607.056} C_VEL
LIN {X 0,Y 509.875,Z 254.593,A -85,B 0,C 180,E1 -5609.75,E2 -5609.75} C_VEL
LIN {X 0,Y 509.871,Z 254.586,A -85,B 0,C 180,E1 -5612.775,E2 -5612.775} C_VEL
LIN {X 0,Y 509.837,Z 254.595,A -85,B 0,C 180,E1 -5615.582,E2 -5615.582} C_VEL
LIN {X 0,Y 509.846,Z 254.6,A -85,B 0,C 180,E1 -5618.339,E2 -5618.339} C_VEL
LIN {X 0,Y 509.861,Z 254.584,A -85,B 0,C 180,E1 -5621.425,E2 -5621.425} C_VEL
LIN {X 0,Y 509.853,Z 254.604,A -85,B 0,C 180,E1 -5624.669,E2 -5624.669} C_VEL
LIN {X 0,Y 509.858,Z 254.589,A -85,B 0,C 180,E1 -5628.103,E2 -5628.103} C_VEL
LIN {X 0,Y 509.845,Z 254.603,A -85,B 0,C 180,E1 -5630.648,E2 -5630.648} C_VEL
LIN {X 0,Y 509.828,Z 254.6,A -85,B 0,C 180,E1 -5633.744,E2 -5633.744} C_VEL
LIN {X 0,Y 509.162,Z 254.69,A -85,B 0,C 180,E1 -5634.403,E2 -5634.403} C_VEL
LIN {X 0,Y 506.346,Z 255.039,A -85,B 0,C 180,E1 -5635.475,E2 -5635.475} C_VEL
LIN {X 0,Y 503.954,Z 255.336,A -85,B 0,C 180,E1 -5636.339,E2 -5636.339} C_VEL
LIN {X 0,Y 502.905,Z 255.466,A -85,B 0,C 180,E1 -5637.005,E2 -5637.005} C_VEL
LIN {X 0,Y 502.807,Z 255.476,A -85,B 0,C 180,E1 -5637.231,E2 -5637.231} C_VEL
LIN {X 0,Y 502.814,Z 255.479,A -85,B 0,C 180,E1 -5640.066,E2 -5640.066} C_VEL
LIN {X 0,Y 502.834,Z 255.466,A -85,B 0,C 180,E1 -5642.534,E2 -5642.534} C_VEL
LIN {X 0,Y 502.846,Z 255.663,A -85,B 0,C 180,E1 -5645.523,E2 -5645.523} C_VEL
LIN {X 0,Y 504.759,Z 265.119,A -85,B 0,C 180,E1 -5647.271,E2 -5647.271} C_VEL
LIN {X 0,Y 504.697,Z 271.467,A -85,B 0,C 180,E1 -5648.345,E2 -5648.345} C_VEL
LIN {X 0,Y 504.142,Z 286.962,A -85,B 0,C 180,E1 -5650.877,E2 -5650.877} C_VEL
LIN {X 0,Y 506.962,Z 302.085,A -85,B 0,C 180,E1 -5651.234,E2 -5651.234} C_VEL
LIN {X 0,Y 506.105,Z 423.487,A -85,B 0,C 180,E1 -5652.994,E2 -5652.994} C_VEL
LIN {X 0,Y 505.773,Z 438.007,A -85,B 0,C 180,E1 -5653.363,E2 -5653.363} C_VEL
LIN {X 0,Y 505.475,Z 452.299,A -85,B 0,C 180,E1 -5653.907,E2 -5653.907} C_VEL
LIN {X 0,Y 505.068,Z 465.312,A -85,B 0,C 180,E1 -5654.567,E2 -5654.567} C_VEL
LIN {X 0,Y 504.534,Z 477.908,A -85,B 0,C 180,E1 -5655.376,E2 -5655.376} C_VEL
LIN {X 0,Y 504.052,Z 489.38,A -85,B 0,C 180,E1 -5656.289,E2 -5656.289} C_VEL
LIN {X 0,Y 503.572,Z 500.102,A -85,B 0,C 180,E1 -5657.323,E2 -5657.323} C_VEL
LIN {X 0,Y 503.227,Z 510.356,A -85,B 0,C 180,E1 -5658.521,E2 -5658.521} C_VEL
LIN {X 0,Y 502.822,Z 518.976,A -85,B 0,C 180,E1 -5659.735,E2 -5659.735} C_VEL
LIN {X 0,Y 502.535,Z 527.241,A -85,B 0,C 180,E1 -5661.151,E2 -5661.151} C_VEL
LIN {X 0,Y 502.352,Z 532.997,A -85,B 0,C 180,E1 -5662.363,E2 -5662.363} C_VEL
LIN {X 0,Y 502.235,Z 537.734,A -85,B 0,C 180,E1 -5663.572,E2 -5663.572} C_VEL
LIN {X 0,Y 502.176,Z 541.578,A -85,B 0,C 180,E1 -5664.781,E2 -5664.781} C_VEL
LIN {X 0,Y 502.146,Z 544.527,A -85,B 0,C 180,E1 -5665.987,E2 -5665.987} C_VEL
LIN {X 0,Y 502.09,Z 547.243,A -85,B 0,C 180,E1 -5667.593,E2 -5667.593} C_VEL
LIN {X 0,Y 501.987,Z 548.608,A -85,B 0,C 180,E1 -5669.198,E2 -5669.198} C_VEL
LIN {X 0,Y 501.988,Z 548.65,A -85,B 0,C 180,E1 -5670.802,E2 -5670.802} C_VEL
LIN {X 0,Y 502.09,Z 547.365,A -85,B 0,C 180,E1 -5672.407,E2 -5672.407} C_VEL
LIN {X 0,Y 502.146,Z 544.723,A -85,B 0,C 180,E1 -5674.013,E2 -5674.013} C_VEL
LIN {X 0,Y 502.24,Z 540.657,A -85,B 0,C 180,E1 -5675.621,E2 -5675.621} C_VEL
LIN {X 0,Y 502.305,Z 535.039,A -85,B 0,C 180,E1 -5677.234,E2 -5677.234} C_VEL
LIN {X 0,Y 502.516,Z 528.696,A -85,B 0,C 180,E1 -5678.647,E2 -5678.647} C_VEL
LIN {X 0,Y 502.736,Z 520.809,A -85,B 0,C 180,E1 -5680.063,E2 -5680.063} C_VEL
LIN {X 0,Y 503.125,Z 512.558,A -85,B 0,C 180,E1 -5681.277,E2 -5681.277} C_VEL
LIN {X 0,Y 503.494,Z 502.621,A -85,B 0,C 180,E1 -5682.494,E2 -5682.494} C_VEL
LIN {X 0,Y 503.963,Z 491.555,A -85,B 0,C 180,E1 -5683.611,E2 -5683.611} C_VEL
LIN {X 0,Y 504.419,Z 480.542,A -85,B 0,C 180,E1 -5684.524,E2 -5684.524} C_VEL
LIN {X 0,Y 504.963,Z 468.593,A -85,B 0,C 180,E1 -5685.333,E2 -5685.333} C_VEL
LIN {X 0,Y 505.386,Z 455.4,A -85,B 0,C 180,E1 -5686.044,E2 -5686.044} C_VEL
LIN {X 0,Y 505.755,Z 441.07,A -85,B 0,C 180,E1 -5686.624,E2 -5686.624} C_VEL
LIN {X 0,Y 506.044,Z 427.482,A -85,B 0,C 180,E1 -5687.008,E2 -5687.008} C_VEL
LIN {X 0,Y 506.23,Z 407.685,A -85,B 0,C 180,E1 -5687.34,E2 -5687.34} C_VEL
LIN {X 0,Y 506.942,Z 301.136,A -85,B 0,C 180,E1 -5688.871,E2 -5688.871} C_VEL
LIN {X 0,Y 504.175,Z 287.048,A -85,B 0,C 180,E1 -5689.207,E2 -5689.207} C_VEL
LIN {X 0,Y 504.38,Z 279.629,A -85,B 0,C 180,E1 -5690.386,E2 -5690.386} C_VEL
LIN {X 0,Y 504.852,Z 265.654,A -85,B 0,C 180,E1 -5692.724,E2 -5692.724} C_VEL
LIN {X 0,Y 502.821,Z 255.577,A -85,B 0,C 180,E1 -5694.606,E2 -5694.606} C_VEL
LIN {X 0,Y 502.834,Z 255.467,A -85,B 0,C 180,E1 -5697.466,E2 -5697.466} C_VEL
LIN {X 0,Y 502.808,Z 255.478,A -85,B 0,C 180,E1 -5700.21,E2 -5700.21} C_VEL
LIN {X 0,Y 502.83,Z 255.474,A -85,B 0,C 180,E1 -5703.03,E2 -5703.03} C_VEL
LIN {X 0,Y 502.779,Z 255.482,A -85,B 0,C 180,E1 -5705.95,E2 -5705.95} C_VEL
LIN {X 0,Y 502.799,Z 255.475,A -85,B 0,C 180,E1 -5708.975,E2 -5708.975} C_VEL
LIN {X 0,Y 502.827,Z 255.464,A -85,B 0,C 180,E1 -5712.135,E2 -5712.135} C_VEL
LIN {X 0,Y 502.797,Z 255.482,A -85,B 0,C 180,E1 -5715.467,E2 -5715.467} C_VEL
LIN {X 0,Y 502.821,Z 255.463,A -85,B 0,C 180,E1 -5719.003,E2 -5719.003} C_VEL
LIN {X 0,Y 502.789,Z 255.478,A -85,B 0,C 180,E1 -5722.045,E2 -5722.045} C_VEL
LIN {X 0,Y 502.804,Z 255.473,A -85,B 0,C 180,E1 -5725.034,E2 -5725.034} C_VEL
LIN {X 0,Y 502.781,Z 255.469,A -85,B 0,C 180,E1 -5727.915,E2 -5727.915} C_VEL
LIN {X 0,Y 502.832,Z 255.474,A -85,B 0,C 180,E1 -5730.713,E2 -5730.713} C_VEL
LIN {X 0,Y 502.855,Z 255.466,A -85,B 0,C 180,E1 -5733.439,E2 -5733.439} C_VEL
LIN {X 0,Y 502.783,Z 255.477,A -85,B 0,C 180,E1 -5736.086,E2 -5736.086} C_VEL
LIN {X 0,Y 502.775,Z 255.481,A -85,B 0,C 180,E1 -5738.688,E2 -5738.688} C_VEL
LIN {X 0,Y 502.822,Z 255.476,A -85,B 0,C 180,E1 -5741.248,E2 -5741.248} C_VEL
LIN {X 0,Y 502.815,Z 255.47,A -85,B 0,C 180,E1 -5743.767,E2 -5743.767} C_VEL
LIN {X 0,Y 502.827,Z 255.469,A -85,B 0,C 180,E1 -5746.254,E2 -5746.254} C_VEL
LIN {X 0,Y 502.873,Z 255.473,A -85,B 0,C 180,E1 -5748.717,E2 -5748.717} C_VEL
LIN {X 0,Y 502.893,Z 255.458,A -85,B 0,C 180,E1 -5751.966,E2 -5751.966} C_VEL
LIN {X 0,Y 502.939,Z 255.462,A -85,B 0,C 180,E1 -5754.386,E2 -5754.386} C_VEL
LIN {X 0,Y 503.016,Z 255.44,A -85,B 0,C 180,E1 -5757.598,E2 -5757.598} C_VEL
LIN {X 0,Y 503.017,Z 255.448,A -85,B 0,C 180,E1 -5760,E2 -5760} C_VEL
LIN {X 0,Y 503.016,Z 255.453,A -85,B 0,C 180,E1 -5762.402,E2 -5762.402} C_VEL
LIN {X 0,Y 502.931,Z 255.456,A -85,B 0,C 180,E1 -5765.614,E2 -5765.614} C_VEL
LIN {X 0,Y 502.893,Z 255.467,A -85,B 0,C 180,E1 -5768.033,E2 -5768.033} C_VEL
LIN {X 0,Y 502.868,Z 255.463,A -85,B 0,C 180,E1 -5771.283,E2 -5771.283} C_VEL
LIN {X 0,Y 502.836,Z 255.472,A -85,B 0,C 180,E1 -5774.571,E2 -5774.571} C_VEL
LIN {X 0,Y 502.853,Z 255.469,A -85,B 0,C 180,E1 -5777.907,E2 -5777.907} C_VEL
LIN {X 0,Y 502.82,Z 255.473,A -85,B 0,C 180,E1 -5780.537,E2 -5780.537} C_VEL
LIN {X 0,Y 502.788,Z 255.474,A -85,B 0,C 180,E1 -5783.041,E2 -5783.041} C_VEL
LIN {X 0,Y 502.832,Z 255.474,A -85,B 0,C 180,E1 -5785.676,E2 -5785.676} C_VEL
LIN {X 0,Y 502.835,Z 255.474,A -85,B 0,C 180,E1 -5788.373,E2 -5788.373} C_VEL
LIN {X 0,Y 502.79,Z 255.478,A -85,B 0,C 180,E1 -5791.5,E2 -5791.5} C_VEL
LIN {X 0,Y 502.799,Z 255.462,A -85,B 0,C 180,E1 -5794.445,E2 -5794.445} C_VEL
LIN {X 0,Y 502.775,Z 255.476,A -85,B 0,C 180,E1 -5797.179,E2 -5797.179} C_VEL
LIN {X 0,Y 502.783,Z 255.479,A -85,B 0,C 180,E1 -5800.016,E2 -5800.016} C_VEL
LIN {X 0,Y 502.797,Z 255.478,A -85,B 0,C 180,E1 -5802.2,E2 -5802.2} C_VEL
LIN {X 0,Y 502.796,Z 255.48,A -85,B 0,C 180,E1 -5805.469,E2 -5805.469} C_VEL
LIN {X 0,Y 502.826,Z 255.467,A -85,B 0,C 180,E1 -5807.865,E2 -5807.865} C_VEL
LIN {X 0,Y 502.806,Z 255.477,A -85,B 0,C 180,E1 -5811.025,E2 -5811.025} C_VEL
LIN {X 0,Y 502.772,Z 255.481,A -85,B 0,C 180,E1 -5814.17,E2 -5814.17} C_VEL
LIN {X 0,Y 502.83,Z 255.47,A -85,B 0,C 180,E1 -5816.994,E2 -5816.994} C_VEL
LIN {X 0,Y 502.813,Z 255.459,A -85,B 0,C 180,E1 -5820.066,E2 -5820.066} C_VEL
LIN {X 0,Y 502.833,Z 255.476,A -85,B 0,C 180,E1 -5822.534,E2 -5822.534} C_VEL
LIN {X 0,Y 502.881,Z 255.569,A -85,B 0,C 180,E1 -5824.327,E2 -5824.327} C_VEL
LIN {X 0,Y 504.22,Z 262.017,A -85,B 0,C 180,E1 -5825.502,E2 -5825.502} C_VEL
LIN {X 0,Y 505.031,Z 266.061,A -85,B 0,C 180,E1 -5826.2,E2 -5826.2} C_VEL
LIN {X 0,Y 504.834,Z 274.143,A -85,B 0,C 180,E1 -5827.491,E2 -5827.491} C_VEL
LIN {X 0,Y 504.239,Z 290.282,A -85,B 0,C 180,E1 -5830.034,E2 -5830.034} C_VEL
LIN {X 0,Y 504.182,Z 295.521,A -85,B 0,C 180,E1 -5830.826,E2 -5830.826} C_VEL
LIN {X 0,Y 506.981,Z 311.361,A -85,B 0,C 180,E1 -5831.194,E2 -5831.194} C_VEL
LIN {X 0,Y 506.075,Z 433.444,A -85,B 0,C 180,E1 -5832.967,E2 -5832.967} C_VEL
LIN {X 0,Y 505.74,Z 447.735,A -85,B 0,C 180,E1 -5833.338,E2 -5833.338} C_VEL
LIN {X 0,Y 505.401,Z 461.269,A -85,B 0,C 180,E1 -5833.853,E2 -5833.853} C_VEL
LIN {X 0,Y 505.022,Z 473.444,A -85,B 0,C 180,E1 -5834.462,E2 -5834.462} C_VEL
LIN {X 0,Y 504.472,Z 486.255,A -85,B 0,C 180,E1 -5835.271,E2 -5835.271} C_VEL
LIN {X 0,Y 504.021,Z 497.902,A -85,B 0,C 180,E1 -5836.185,E2 -5836.185} C_VEL
LIN {X 0,Y 503.52,Z 509.55,A -85,B 0,C 180,E1 -5837.301,E2 -5837.301} C_VEL
LIN {X 0,Y 503.182,Z 519.963,A -85,B 0,C 180,E1 -5838.52,E2 -5838.52} C_VEL
LIN {X 0,Y 502.767,Z 528.554,A -85,B 0,C 180,E1 -5839.734,E2 -5839.734} C_VEL
LIN {X 0,Y 502.507,Z 536.78,A -85,B 0,C 180,E1 -5841.15,E2 -5841.15} C_VEL
LIN {X 0,Y 502.318,Z 542.537,A -85,B 0,C 180,E1 -5842.362,E2 -5842.362} C_VEL
LIN {X 0,Y 502.234,Z 547.254,A -85,B 0,C 180,E1 -5843.573,E2 -5843.573} C_VEL
LIN {X 0,Y 502.17,Z 551.074,A -85,B 0,C 180,E1 -5844.781,E2 -5844.781} C_VEL
LIN {X 0,Y 502.113,Z 554.017,A -85,B 0,C 180,E1 -5845.987,E2 -5845.987} C_VEL
LIN {X 0,Y 502.064,Z 556.711,A -85,B 0,C 180,E1 -5847.593,E2 -5847.593} C_VEL
LIN {X 0,Y 501.988,Z 558.045,A -85,B 0,C 180,E1 -5849.198,E2 -5849.198} C_VEL
LIN {X 0,Y 501.988,Z 558.045,A -85,B 0,C 180,E1 -5850.802,E2 -5850.802} C_VEL
LIN {X 0,Y 502.064,Z 556.713,A -85,B 0,C 180,E1 -5852.407,E2 -5852.407} C_VEL
LIN {X 0,Y 502.113,Z 554.021,A -85,B 0,C 180,E1 -5854.013,E2 -5854.013} C_VEL
LIN {X 0,Y 502.21,Z 549.892,A -85,B 0,C 180,E1 -5855.622,E2 -5855.622} C_VEL
LIN {X 0,Y 502.253,Z 544.203,A -85,B 0,C 180,E1 -5857.235,E2 -5857.235} C_VEL
LIN {X 0,Y 502.473,Z 537.79,A -85,B 0,C 180,E1 -5858.648,E2 -5858.648} C_VEL
LIN {X 0,Y 502.709,Z 529.82,A -85,B 0,C 180,E1 -5860.064,E2 -5860.064} C_VEL
LIN {X 0,Y 503.079,Z 521.484,A -85,B 0,C 180,E1 -5861.278,E2 -5861.278} C_VEL
LIN {X 0,Y 503.509,Z 510.81,A -85,B 0,C 180,E1 -5862.566,E2 -5862.566} C_VEL
LIN {X 0,Y 503.917,Z 500.248,A -85,B 0,C 180,E1 -5863.612,E2 -5863.612} C_VEL
LIN {X 0,Y 504.357,Z 489.109,A -85,B 0,C 180,E1 -5864.526,E2 -5864.526} C_VEL
LIN {X 0,Y 504.898,Z 476.978,A -85,B 0,C 180,E1 -5865.335,E2 -5865.335} C_VEL
LIN {X 0,Y 505.38,Z 463.517,A -85,B 0,C 180,E1 -5866.044,E2 -5866.044} C_VEL
LIN {X 0,Y 505.718,Z 449.705,A -85,B 0,C 180,E1 -5866.595,E2 -5866.595} C_VEL
LIN {X 0,Y 506.032,Z 435.716,A -85,B 0,C 180,E1 -5866.983,E2 -5866.983} C_VEL
LIN {X 0,Y 506.233,Z 415.439,A -85,B 0,C 180,E1 -5867.314,E2 -5867.314} C_VEL
LIN {X 0,Y 506.878,Z 310.456,A -85,B 0,C 180,E1 -5868.823,E2 -5868.823} C_VEL
LIN {X 0,Y 504.18,Z 295.664,A -85,B 0,C 180,E1 -5869.164,E2 -5869.164} C_VEL
LIN {X 0,Y 504.738,Z 276.83,A -85,B 0,C 180,E1 -5872.083,E2 -5872.083} C_VEL
LIN {X 0,Y 505.141,Z 267.963,A -85,B 0,C 180,E1 -5873.488,E2 -5873.488} C_VEL
LIN {X 0,Y 504.501,Z 263.36,A -85,B 0,C 180,E1 -5874.264,E2 -5874.264} C_VEL
LIN {X 0,Y 502.905,Z 255.726,A -85,B 0,C 180,E1 -5875.618,E2 -5875.618} C_VEL
LIN {X 0,Y 502.863,Z 255.457,A -85,B 0,C 180,E1 -5876.119,E2 -5876.119} C_VEL
LIN {X 0,Y 502.823,Z 255.459,A -85,B 0,C 180,E1 -5879.287,E2 -5879.287} C_VEL
LIN {X 0,Y 502.783,Z 255.48,A -85,B 0,C 180,E1 -5882.084,E2 -5882.084} C_VEL
LIN {X 0,Y 502.797,Z 255.479,A -85,B 0,C 180,E1 -5884.965,E2 -5884.965} C_VEL
LIN {X 0,Y 502.79,Z 255.474,A -85,B 0,C 180,E1 -5887.953,E2 -5887.953} C_VEL
LIN {X 0,Y 502.816,Z 255.466,A -85,B 0,C 180,E1 -5891.065,E2 -5891.065} C_VEL
LIN {X 0,Y 502.778,Z 255.477,A -85,B 0,C 180,E1 -5893.375,E2 -5893.375} C_VEL
LIN {X 0,Y 502.785,Z 255.477,A -85,B 0,C 180,E1 -5895.661,E2 -5895.661} C_VEL
LIN {X 0,Y 502.814,Z 255.47,A -85,B 0,C 180,E1 -5899.004,E2 -5899.004} C_VEL
LIN {X 0,Y 502.789,Z 255.483,A -85,B 0,C 180,E1 -5902.046,E2 -5902.046} C_VEL
LIN {X 0,Y 502.803,Z 255.459,A -85,B 0,C 180,E1 -5905.035,E2 -5905.035} C_VEL
LIN {X 0,Y 502.782,Z 255.475,A -85,B 0,C 180,E1 -5907.915,E2 -5907.915} C_VEL
LIN {X 0,Y 502.833,Z 255.471,A -85,B 0,C 180,E1 -5910.713,E2 -5910.713} C_VEL
LIN {X 0,Y 502.874,Z 255.464,A -85,B 0,C 180,E1 -5913.434,E2 -5913.434} C_VEL
LIN {X 0,Y 502.784,Z 255.48,A -85,B 0,C 180,E1 -5916.086,E2 -5916.086} C_VEL
LIN {X 0,Y 502.775,Z 255.476,A -85,B 0,C 180,E1 -5918.689,E2 -5918.689} C_VEL
LIN {X 0,Y 502.822,Z 255.473,A -85,B 0,C 180,E1 -5921.248,E2 -5921.248} C_VEL
LIN {X 0,Y 502.816,Z 255.474,A -85,B 0,C 180,E1 -5923.767,E2 -5923.767} C_VEL
LIN {X 0,Y 502.824,Z 255.474,A -85,B 0,C 180,E1 -5926.255,E2 -5926.255} C_VEL
LIN {X 0,Y 502.869,Z 255.462,A -85,B 0,C 180,E1 -5928.717,E2 -5928.717} C_VEL
LIN {X 0,Y 502.893,Z 255.467,A -85,B 0,C 180,E1 -5931.967,E2 -5931.967} C_VEL
LIN {X 0,Y 502.931,Z 255.456,A -85,B 0,C 180,E1 -5934.386,E2 -5934.386} C_VEL
LIN {X 0,Y 503.016,Z 255.452,A -85,B 0,C 180,E1 -5937.598,E2 -5937.598} C_VEL
LIN {X 0,Y 503.018,Z 255.448,A -85,B 0,C 180,E1 -5940,E2 -5940} C_VEL
LIN {X 0,Y 503.017,Z 255.44,A -85,B 0,C 180,E1 -5942.402,E2 -5942.402} C_VEL
LIN {X 0,Y 502.939,Z 255.463,A -85,B 0,C 180,E1 -5945.614,E2 -5945.614} C_VEL
LIN {X 0,Y 502.893,Z 255.459,A -85,B 0,C 180,E1 -5948.034,E2 -5948.034} C_VEL
LIN {X 0,Y 502.869,Z 255.473,A -85,B 0,C 180,E1 -5951.283,E2 -5951.283} C_VEL
LIN {X 0,Y 502.837,Z 255.467,A -85,B 0,C 180,E1 -5954.571,E2 -5954.571} C_VEL
LIN {X 0,Y 502.854,Z 255.469,A -85,B 0,C 180,E1 -5957.907,E2 -5957.907} C_VEL
LIN {X 0,Y 502.821,Z 255.47,A -85,B 0,C 180,E1 -5960.537,E2 -5960.537} C_VEL
LIN {X 0,Y 502.787,Z 255.483,A -85,B 0,C 180,E1 -5963.041,E2 -5963.041} C_VEL
LIN {X 0,Y 502.833,Z 255.467,A -85,B 0,C 180,E1 -5965.676,E2 -5965.676} C_VEL
LIN {X 0,Y 502.836,Z 255.471,A -85,B 0,C 180,E1 -5968.373,E2 -5968.373} C_VEL
LIN {X 0,Y 502.791,Z 255.469,A -85,B 0,C 180,E1 -5971.5,E2 -5971.5} C_VEL
LIN {X 0,Y 502.801,Z 255.462,A -85,B 0,C 180,E1 -5974.445,E2 -5974.445} C_VEL
LIN {X 0,Y 502.776,Z 255.482,A -85,B 0,C 180,E1 -5977.179,E2 -5977.179} C_VEL
LIN {X 0,Y 502.812,Z 255.47,A -85,B 0,C 180,E1 -5980.013,E2 -5980.013} C_VEL
LIN {X 0,Y 502.77,Z 255.479,A -85,B 0,C 180,E1 -5983.232,E2 -5983.232} C_VEL
LIN {X 0,Y 502.787,Z 255.476,A -85,B 0,C 180,E1 -5985.662,E2 -5985.662} C_VEL
LIN {X 0,Y 502.827,Z 255.462,A -85,B 0,C 180,E1 -5987.865,E2 -5987.865} C_VEL
LIN {X 0,Y 502.8,Z 255.475,A -85,B 0,C 180,E1 -5991.025,E2 -5991.025} C_VEL
LIN {X 0,Y 502.781,Z 255.481,A -85,B 0,C 180,E1 -5994.168,E2 -5994.168} C_VEL
LIN {X 0,Y 502.807,Z 255.476,A -85,B 0,C 180,E1 -5997.231,E2 -5997.231} C_VEL
LIN {X 0,Y 502.106,Z 255.566,A -85,B 0,C 180,E1 -5997.899,E2 -5997.899} C_VEL
LIN {X 0,Y 499.242,Z 255.923,A -85,B 0,C 180,E1 -5998.985,E2 -5998.985} C_VEL
LIN {X 0,Y 496.847,Z 256.221,A -85,B 0,C 180,E1 -5999.86,E2 -5999.86} C_VEL
LIN {X 0,Y 495.831,Z 256.345,A -85,B 0,C 180,E1 -6000.536,E2 -6000.536} C_VEL
LIN {X 0,Y 495.753,Z 256.351,A -85,B 0,C 180,E1 -6000.764,E2 -6000.764} C_VEL
LIN {X 0,Y 495.824,Z 256.349,A -85,B 0,C 180,E1 -6003.251,E2 -6003.251} C_VEL
LIN {X 0,Y 495.811,Z 256.55,A -85,B 0,C 180,E1 -6005.299,E2 -6005.299} C_VEL
LIN {X 0,Y 497.976,Z 267.716,A -85,B 0,C 180,E1 -6007.383,E2 -6007.383} C_VEL
LIN {X 0,Y 497.246,Z 286.434,A -85,B 0,C 180,E1 -6010.53,E2 -6010.53} C_VEL
LIN {X 0,Y 497.276,Z 287.233,A -85,B 0,C 180,E1 -6010.615,E2 -6010.615} C_VEL
LIN {X 0,Y 500.266,Z 303.047,A -85,B 0,C 180,E1 -6010.986,E2 -6010.986} C_VEL
LIN {X 0,Y 499.346,Z 423.582,A -85,B 0,C 180,E1 -6012.756,E2 -6012.756} C_VEL
LIN {X 0,Y 499.016,Z 437.869,A -85,B 0,C 180,E1 -6013.123,E2 -6013.123} C_VEL
LIN {X 0,Y 498.697,Z 451.25,A -85,B 0,C 180,E1 -6013.629,E2 -6013.629} C_VEL
LIN {X 0,Y 498.28,Z 463.625,A -85,B 0,C 180,E1 -6014.246,E2 -6014.246} C_VEL
LIN {X 0,Y 497.728,Z 476.56,A -85,B 0,C 180,E1 -6015.067,E2 -6015.067} C_VEL
LIN {X 0,Y 497.192,Z 488.283,A -85,B 0,C 180,E1 -6015.992,E2 -6015.992} C_VEL
LIN {X 0,Y 496.683,Z 499.104,A -85,B 0,C 180,E1 -6017.03,E2 -6017.03} C_VEL
LIN {X 0,Y 496.288,Z 509.034,A -85,B 0,C 180,E1 -6018.18,E2 -6018.18} C_VEL
LIN {X 0,Y 495.867,Z 517.696,A -85,B 0,C 180,E1 -6019.383,E2 -6019.383} C_VEL
LIN {X 0,Y 495.548,Z 526.208,A -85,B 0,C 180,E1 -6020.819,E2 -6020.819} C_VEL
LIN {X 0,Y 495.293,Z 533.067,A -85,B 0,C 180,E1 -6022.253,E2 -6022.253} C_VEL
LIN {X 0,Y 495.151,Z 538.707,A -85,B 0,C 180,E1 -6023.741,E2 -6023.741} C_VEL
LIN {X 0,Y 495.032,Z 542.709,A -85,B 0,C 180,E1 -6025.114,E2 -6025.114} C_VEL
LIN {X 0,Y 495.038,Z 546.125,A -85,B 0,C 180,E1 -6026.745,E2 -6026.745} C_VEL
LIN {X 0,Y 494.961,Z 548.158,A -85,B 0,C 180,E1 -6028.373,E2 -6028.373} C_VEL
LIN {X 0,Y 494.897,Z 548.861,A -85,B 0,C 180,E1 -6030,E2 -6030} C_VEL
LIN {X 0,Y 494.96,Z 548.24,A -85,B 0,C 180,E1 -6031.627,E2 -6031.627} C_VEL
LIN {X 0,Y 495.037,Z 546.281,A -85,B 0,C 180,E1 -6033.255,E2 -6033.255} C_VEL
LIN {X 0,Y 495.032,Z 542.94,A -85,B 0,C 180,E1 -6034.886,E2 -6034.886} C_VEL
LIN {X 0,Y 495.163,Z 538.972,A -85,B 0,C 180,E1 -6036.273,E2 -6036.273} C_VEL
LIN {X 0,Y 495.287,Z 533.464,A -85,B 0,C 180,E1 -6037.747,E2 -6037.747} C_VEL
LIN {X 0,Y 495.545,Z 526.695,A -85,B 0,C 180,E1 -6039.181,E2 -6039.181} C_VEL
LIN {X 0,Y 495.839,Z 518.286,A -85,B 0,C 180,E1 -6040.618,E2 -6040.618} C_VEL
LIN {X 0,Y 496.268,Z 508.565,A -85,B 0,C 180,E1 -6041.97,E2 -6041.97} C_VEL
LIN {X 0,Y 496.69,Z 498.877,A -85,B 0,C 180,E1 -6043.085,E2 -6043.085} C_VEL
LIN {X 0,Y 497.212,Z 488.123,A -85,B 0,C 180,E1 -6044.112,E2 -6044.112} C_VEL
LIN {X 0,Y 497.73,Z 476.359,A -85,B 0,C 180,E1 -6045.037,E2 -6045.037} C_VEL
LIN {X 0,Y 498.288,Z 463.379,A -85,B 0,C 180,E1 -6045.859,E2 -6045.859} C_VEL
LIN {X 0,Y 498.738,Z 449.779,A -85,B 0,C 180,E1 -6046.527,E2 -6046.527} C_VEL
LIN {X 0,Y 499.077,Z 435.855,A -85,B 0,C 180,E1 -6047.029,E2 -6047.029} C_VEL
LIN {X 0,Y 499.388,Z 421.248,A -85,B 0,C 180,E1 -6047.374,E2 -6047.374} C_VEL
LIN {X 0,Y 500.292,Z 302.537,A -85,B 0,C 180,E1 -6049.111,E2 -6049.111} C_VEL
LIN {X 0,Y 497.267,Z 287.174,A -85,B 0,C 180,E1 -6049.481,E2 -6049.481} C_VEL
LIN {X 0,Y 497.48,Z 279.688,A -85,B 0,C 180,E1 -6050.681,E2 -6050.681} C_VEL
LIN {X 0,Y 497.922,Z 266.977,A -85,B 0,C 180,E1 -6052.839,E2 -6052.839} C_VEL
LIN {X 0,Y 495.777,Z 256.458,A -85,B 0,C 180,E1 -6054.833,E2 -6054.833} C_VEL
LIN {X 0,Y 495.814,Z 256.349,A -85,B 0,C 180,E1 -6056.973,E2 -6056.973} C_VEL
LIN {X 0,Y 495.764,Z 256.356,A -85,B 0,C 180,E1 -6060.146,E2 -6060.146} C_VEL
LIN {X 0,Y 495.792,Z 256.353,A -85,B 0,C 180,E1 -6063.244,E2 -6063.244} C_VEL
LIN {X 0,Y 495.724,Z 256.36,A -85,B 0,C 180,E1 -6066.089,E2 -6066.089} C_VEL
LIN {X 0,Y 495.761,Z 256.35,A -85,B 0,C 180,E1 -6068.767,E2 -6068.767} C_VEL
LIN {X 0,Y 495.774,Z 256.345,A -85,B 0,C 180,E1 -6071.778,E2 -6071.778} C_VEL
LIN {X 0,Y 495.745,Z 256.358,A -85,B 0,C 180,E1 -6075.139,E2 -6075.139} C_VEL
LIN {X 0,Y 495.755,Z 256.34,A -85,B 0,C 180,E1 -6078.219,E2 -6078.219} C_VEL
LIN {X 0,Y 495.764,Z 256.356,A -85,B 0,C 180,E1 -6081.23,E2 -6081.23} C_VEL
LIN {X 0,Y 495.752,Z 256.351,A -85,B 0,C 180,E1 -6084.462,E2 -6084.462} C_VEL
LIN {X 0,Y 495.763,Z 256.343,A -85,B 0,C 180,E1 -6087.405,E2 -6087.405} C_VEL
LIN {X 0,Y 495.775,Z 256.35,A -85,B 0,C 180,E1 -6090.254,E2 -6090.254} C_VEL
LIN {X 0,Y 495.816,Z 256.345,A -85,B 0,C 180,E1 -6093.25,E2 -6093.25} C_VEL
LIN {X 0,Y 495.744,Z 256.354,A -85,B 0,C 180,E1 -6095.724,E2 -6095.724} C_VEL
LIN {X 0,Y 495.734,Z 256.355,A -85,B 0,C 180,E1 -6098.371,E2 -6098.371} C_VEL
LIN {X 0,Y 495.777,Z 256.356,A -85,B 0,C 180,E1 -6100.971,E2 -6100.971} C_VEL
LIN {X 0,Y 495.772,Z 256.348,A -85,B 0,C 180,E1 -6103.53,E2 -6103.53} C_VEL
LIN {X 0,Y 495.788,Z 256.344,A -85,B 0,C 180,E1 -6106.055,E2 -6106.055} C_VEL
LIN {X 0,Y 495.846,Z 256.347,A -85,B 0,C 180,E1 -6108.555,E2 -6108.555} C_VEL
LIN {X 0,Y 495.864,Z 256.333,A -85,B 0,C 180,E1 -6111.852,E2 -6111.852} C_VEL
LIN {X 0,Y 495.895,Z 256.339,A -85,B 0,C 180,E1 -6114.306,E2 -6114.306} C_VEL
LIN {X 0,Y 495.985,Z 256.315,A -85,B 0,C 180,E1 -6117.564,E2 -6117.564} C_VEL
LIN {X 0,Y 495.988,Z 256.324,A -85,B 0,C 180,E1 -6120,E2 -6120} C_VEL
LIN {X 0,Y 495.985,Z 256.328,A -85,B 0,C 180,E1 -6122.436,E2 -6122.436} C_VEL
LIN {X 0,Y 495.888,Z 256.334,A -85,B 0,C 180,E1 -6125.694,E2 -6125.694} C_VEL
LIN {X 0,Y 495.864,Z 256.344,A -85,B 0,C 180,E1 -6128.148,E2 -6128.148} C_VEL
LIN {X 0,Y 495.842,Z 256.338,A -85,B 0,C 180,E1 -6131.445,E2 -6131.445} C_VEL
LIN {X 0,Y 495.781,Z 256.349,A -85,B 0,C 180,E1 -6134.783,E2 -6134.783} C_VEL
LIN {X 0,Y 495.779,Z 256.345,A -85,B 0,C 180,E1 -6137.319,E2 -6137.319} C_VEL
LIN {X 0,Y 495.763,Z 256.356,A -85,B 0,C 180,E1 -6139.891,E2 -6139.891} C_VEL
LIN {X 0,Y 495.757,Z 256.35,A -85,B 0,C 180,E1 -6142.863,E2 -6142.863} C_VEL
LIN {X 0,Y 495.783,Z 256.353,A -85,B 0,C 180,E1 -6146.068,E2 -6146.068} C_VEL
LIN {X 0,Y 495.773,Z 256.35,A -85,B 0,C 180,E1 -6148.815,E2 -6148.815} C_VEL
LIN {X 0,Y 495.752,Z 256.357,A -85,B 0,C 180,E1 -6151.727,E2 -6151.727} C_VEL
LIN {X 0,Y 495.769,Z 256.335,A -85,B 0,C 180,E1 -6154.696,E2 -6154.696} C_VEL
LIN {X 0,Y 495.725,Z 256.358,A -85,B 0,C 180,E1 -6157.562,E2 -6157.562} C_VEL
LIN {X 0,Y 495.761,Z 256.349,A -85,B 0,C 180,E1 -6160.7,E2 -6160.7} C_VEL
LIN {X 0,Y 495.729,Z 256.359,A -85,B 0,C 180,E1 -6164.002,E2 -6164.002} C_VEL
LIN {X 0,Y 495.76,Z 256.353,A -85,B 0,C 180,E1 -6167.122,E2 -6167.122} C_VEL
LIN {X 0,Y 495.779,Z 256.351,A -85,B 0,C 180,E1 -6170.365,E2 -6170.365} C_VEL
LIN {X 0,Y 495.725,Z 256.356,A -85,B 0,C 180,E1 -6173.457,E2 -6173.457} C_VEL
LIN {X 0,Y 495.757,Z 256.349,A -85,B 0,C 180,E1 -6176.436,E2 -6176.436} C_VEL
LIN {X 0,Y 495.75,Z 256.346,A -85,B 0,C 180,E1 -6179.313,E2 -6179.313} C_VEL
LIN {X 0,Y 495.78,Z 256.355,A -85,B 0,C 180,E1 -6182.109,E2 -6182.109} C_VEL
LIN {X 0,Y 495.851,Z 256.475,A -85,B 0,C 180,E1 -6184.106,E2 -6184.106} C_VEL
LIN {X 0,Y 498.195,Z 268.32,A -85,B 0,C 180,E1 -6186.232,E2 -6186.232} C_VEL
LIN {X 0,Y 497.547,Z 285.82,A -85,B 0,C 180,E1 -6189.045,E2 -6189.045} C_VEL
LIN {X 0,Y 497.233,Z 295.454,A -85,B 0,C 180,E1 -6190.547,E2 -6190.547} C_VEL
LIN {X 0,Y 500.238,Z 312.718,A -85,B 0,C 180,E1 -6190.952,E2 -6190.952} C_VEL
LIN {X 0,Y 499.289,Z 433.38,A -85,B 0,C 180,E1 -6192.728,E2 -6192.728} C_VEL
LIN {X 0,Y 498.937,Z 447.372,A -85,B 0,C 180,E1 -6193.094,E2 -6193.094} C_VEL
LIN {X 0,Y 498.576,Z 461.203,A -85,B 0,C 180,E1 -6193.625,E2 -6193.625} C_VEL
LIN {X 0,Y 498.168,Z 473.378,A -85,B 0,C 180,E1 -6194.243,E2 -6194.243} C_VEL
LIN {X 0,Y 497.562,Z 486.188,A -85,B 0,C 180,E1 -6195.062,E2 -6195.062} C_VEL
LIN {X 0,Y 497.108,Z 497.836,A -85,B 0,C 180,E1 -6195.989,E2 -6195.989} C_VEL
LIN {X 0,Y 496.584,Z 508.602,A -85,B 0,C 180,E1 -6197.027,E2 -6197.027} C_VEL
LIN {X 0,Y 496.195,Z 518.508,A -85,B 0,C 180,E1 -6198.18,E2 -6198.18} C_VEL
LIN {X 0,Y 495.818,Z 527.131,A -85,B 0,C 180,E1 -6199.382,E2 -6199.382} C_VEL
LIN {X 0,Y 495.48,Z 535.625,A -85,B 0,C 180,E1 -6200.818,E2 -6200.818} C_VEL
LIN {X 0,Y 495.238,Z 542.47,A -85,B 0,C 180,E1 -6202.252,E2 -6202.252} C_VEL
LIN {X 0,Y 495.116,Z 548.195,A -85,B 0,C 180,E1 -6203.769,E2 -6203.769} C_VEL
LIN {X 0,Y 495.03,Z 552.073,A -85,B 0,C 180,E1 -6205.114,E2 -6205.114} C_VEL
LIN {X 0,Y 495.033,Z 555.47,A -85,B 0,C 180,E1 -6206.745,E2 -6206.745} C_VEL
LIN {X 0,Y 494.958,Z 557.479,A -85,B 0,C 180,E1 -6208.373,E2 -6208.373} C_VEL
LIN {X 0,Y 494.896,Z 558.145,A -85,B 0,C 180,E1 -6210,E2 -6210} C_VEL
LIN {X 0,Y 494.958,Z 557.481,A -85,B 0,C 180,E1 -6211.627,E2 -6211.627} C_VEL
LIN {X 0,Y 495.033,Z 555.474,A -85,B 0,C 180,E1 -6213.255,E2 -6213.255} C_VEL
LIN {X 0,Y 495.03,Z 552.076,A -85,B 0,C 180,E1 -6214.886,E2 -6214.886} C_VEL
LIN {X 0,Y 495.133,Z 547.29,A -85,B 0,C 180,E1 -6216.49,E2 -6216.49} C_VEL
LIN {X 0,Y 495.238,Z 542.468,A -85,B 0,C 180,E1 -6217.748,E2 -6217.748} C_VEL
LIN {X 0,Y 495.489,Z 535.626,A -85,B 0,C 180,E1 -6219.182,E2 -6219.182} C_VEL
LIN {X 0,Y 495.818,Z 527.13,A -85,B 0,C 180,E1 -6220.618,E2 -6220.618} C_VEL
LIN {X 0,Y 496.203,Z 517.387,A -85,B 0,C 180,E1 -6221.963,E2 -6221.963} C_VEL
LIN {X 0,Y 496.649,Z 507.527,A -85,B 0,C 180,E1 -6223.086,E2 -6223.086} C_VEL
LIN {X 0,Y 497.154,Z 495.484,A -85,B 0,C 180,E1 -6224.218,E2 -6224.218} C_VEL
LIN {X 0,Y 497.764,Z 483.31,A -85,B 0,C 180,E1 -6225.141,E2 -6225.141} C_VEL
LIN {X 0,Y 498.237,Z 471.598,A -85,B 0,C 180,E1 -6225.86,E2 -6225.86} C_VEL
LIN {X 0,Y 498.704,Z 457.905,A -85,B 0,C 180,E1 -6226.517,E2 -6226.517} C_VEL
LIN {X 0,Y 499.063,Z 444.182,A -85,B 0,C 180,E1 -6227.002,E2 -6227.002} C_VEL
LIN {X 0,Y 499.327,Z 430.615,A -85,B 0,C 180,E1 -6227.324,E2 -6227.324} C_VEL
LIN {X 0,Y 500.186,Z 311.5,A -85,B 0,C 180,E1 -6229.068,E2 -6229.068} C_VEL
LIN {X 0,Y 497.247,Z 295.708,A -85,B 0,C 180,E1 -6229.436,E2 -6229.436} C_VEL
LIN {X 0,Y 497.273,Z 291.557,A -85,B 0,C 180,E1 -6230.043,E2 -6230.043} C_VEL
LIN {X 0,Y 497.964,Z 275.424,A -85,B 0,C 180,E1 -6232.618,E2 -6232.618} C_VEL
LIN {X 0,Y 498.196,Z 268.313,A -85,B 0,C 180,E1 -6233.768,E2 -6233.768} C_VEL
LIN {X 0,Y 495.852,Z 256.474,A -85,B 0,C 180,E1 -6235.894,E2 -6235.894} C_VEL
LIN {X 0,Y 495.771,Z 256.342,A -85,B 0,C 180,E1 -6238.814,E2 -6238.814} C_VEL
LIN {X 0,Y 495.754,Z 256.354,A -85,B 0,C 180,E1 -6241.725,E2 -6241.725} C_VEL
LIN {X 0,Y 495.766,Z 256.358,A -85,B 0,C 180,E1 -6244.693,E2 -6244.693} C_VEL
LIN {X 0,Y 495.726,Z 256.352,A -85,B 0,C 180,E1 -6247.561,E2 -6247.561} C_VEL
LIN {X 0,Y 495.763,Z 256.347,A -85,B 0,C 180,E1 -6250.699,E2 -6250.699} C_VEL
LIN {X 0,Y 495.731,Z 256.356,A -85,B 0,C 180,E1 -6253.695,E2 -6253.695} C_VEL
LIN {X 0,Y 495.724,Z 256.361,A -85,B 0,C 180,E1 -6256.305,E2 -6256.305} C_VEL
LIN {X 0,Y 495.762,Z 256.348,A -85,B 0,C 180,E1 -6259.3,E2 -6259.3} C_VEL
LIN {X 0,Y 495.726,Z 256.358,A -85,B 0,C 180,E1 -6262.438,E2 -6262.438} C_VEL
LIN {X 0,Y 495.779,Z 256.334,A -85,B 0,C 180,E1 -6265.457,E2 -6265.457} C_VEL
LIN {X 0,Y 495.753,Z 256.357,A -85,B 0,C 180,E1 -6268.364,E2 -6268.364} C_VEL
LIN {X 0,Y 495.783,Z 256.35,A -85,B 0,C 180,E1 -6271.506,E2 -6271.506} C_VEL
LIN {X 0,Y 495.793,Z 256.352,A -85,B 0,C 180,E1 -6273.932,E2 -6273.932} C_VEL
LIN {X 0,Y 495.758,Z 256.349,A -85,B 0,C 180,E1 -6277.137,E2 -6277.137} C_VEL
LIN {X 0,Y 495.764,Z 256.356,A -85,B 0,C 180,E1 -6280.109,E2 -6280.109} C_VEL
LIN {X 0,Y 495.78,Z 256.345,A -85,B 0,C 180,E1 -6282.681,E2 -6282.681} C_VEL
LIN {X 0,Y 495.782,Z 256.348,A -85,B 0,C 180,E1 -6285.217,E2 -6285.217} C_VEL
LIN {X 0,Y 495.843,Z 256.338,A -85,B 0,C 180,E1 -6288.555,E2 -6288.555} C_VEL
LIN {X 0,Y 495.865,Z 256.344,A -85,B 0,C 180,E1 -6291.852,E2 -6291.852} C_VEL
LIN {X 0,Y 495.888,Z 256.334,A -85,B 0,C 180,E1 -6294.306,E2 -6294.306} C_VEL
LIN {X 0,Y 495.985,Z 256.327,A -85,B 0,C 180,E1 -6297.564,E2 -6297.564} C_VEL
LIN {X 0,Y 495.989,Z 256.324,A -85,B 0,C 180,E1 -6300,E2 -6300} C_VEL
LIN {X 0,Y 495.985,Z 256.315,A -85,B 0,C 180,E1 -6302.436,E2 -6302.436} C_VEL
LIN {X 0,Y 495.895,Z 256.339,A -85,B 0,C 180,E1 -6305.694,E2 -6305.694} C_VEL
LIN {X 0,Y 495.865,Z 256.333,A -85,B 0,C 180,E1 -6308.148,E2 -6308.148} C_VEL
LIN {X 0,Y 495.843,Z 256.348,A -85,B 0,C 180,E1 -6311.445,E2 -6311.445} C_VEL
LIN {X 0,Y 495.782,Z 256.347,A -85,B 0,C 180,E1 -6314.783,E2 -6314.783} C_VEL
LIN {X 0,Y 495.781,Z 256.356,A -85,B 0,C 180,E1 -6317.319,E2 -6317.319} C_VEL
LIN {X 0,Y 495.764,Z 256.348,A -85,B 0,C 180,E1 -6319.891,E2 -6319.891} C_VEL
LIN {X 0,Y 495.754,Z 256.356,A -85,B 0,C 180,E1 -6322.862,E2 -6322.862} C_VEL
LIN {X 0,Y 495.784,Z 256.344,A -85,B 0,C 180,E1 -6326.068,E2 -6326.068} C_VEL
LIN {X 0,Y 495.774,Z 256.356,A -85,B 0,C 180,E1 -6328.815,E2 -6328.815} C_VEL
LIN {X 0,Y 495.753,Z 256.344,A -85,B 0,C 180,E1 -6331.727,E2 -6331.727} C_VEL
LIN {X 0,Y 495.771,Z 256.34,A -85,B 0,C 180,E1 -6334.696,E2 -6334.696} C_VEL
LIN {X 0,Y 495.726,Z 256.357,A -85,B 0,C 180,E1 -6337.562,E2 -6337.562} C_VEL
LIN {X 0,Y 495.774,Z 256.344,A -85,B 0,C 180,E1 -6340.699,E2 -6340.699} C_VEL
LIN {X 0,Y 495.73,Z 256.355,A -85,B 0,C 180,E1 -6344.002,E2 -6344.002} C_VEL
LIN {X 0,Y 495.731,Z 256.348,A -85,B 0,C 180,E1 -6347.119,E2 -6347.119} C_VEL
LIN {X 0,Y 495.757,Z 256.354,A -85,B 0,C 180,E1 -6349.954,E2 -6349.954} C_VEL
LIN {X 0,Y 495.728,Z 256.357,A -85,B 0,C 180,E1 -6352.554,E2 -6352.554} C_VEL
LIN {X 0,Y 495.782,Z 256.347,A -85,B 0,C 180,E1 -6355.458,E2 -6355.458} C_VEL
LIN {X 0,Y 495.756,Z 256.356,A -85,B 0,C 180,E1 -6358.364,E2 -6358.364} C_VEL
LIN {X 0,Y 495.753,Z 256.351,A -85,B 0,C 180,E1 -6360.764,E2 -6360.764} C_VEL
LIN {X 0,Y 495.096,Z 256.429,A -85,B 0,C 180,E1 -6361.444,E2 -6361.444} C_VEL
LIN {X 0,Y 492.239,Z 256.785,A -85,B 0,C 180,E1 -6362.546,E2 -6362.546} C_VEL
LIN {X 0,Y 489.824,Z 257.096,A -85,B 0,C 180,E1 -6363.435,E2 -6363.435} C_VEL
LIN {X 0,Y 488.801,Z 257.22,A -85,B 0,C 180,E1 -6364.121,E2 -6364.121} C_VEL
LIN {X 0,Y 488.725,Z 257.225,A -85,B 0,C 180,E1 -6364.353,E2 -6364.353} C_VEL
LIN {X 0,Y 488.733,Z 257.38,A -85,B 0,C 180,E1 -6365.045,E2 -6365.045} C_VEL
LIN {X 0,Y 491.068,Z 269.048,A -85,B 0,C 180,E1 -6367.269,E2 -6367.269} C_VEL
LIN {X 0,Y 490.359,Z 286.966,A -85,B 0,C 180,E1 -6370.305,E2 -6370.305} C_VEL
LIN {X 0,Y 491.729,Z 294.043,A -85,B 0,C 180,E1 -6370.504,E2 -6370.504} C_VEL
LIN {X 0,Y 493.58,Z 303.817,A -85,B 0,C 180,E1 -6370.728,E2 -6370.728} C_VEL
LIN {X 0,Y 492.593,Z 423.673,A -85,B 0,C 180,E1 -6372.512,E2 -6372.512} C_VEL
LIN {X 0,Y 492.244,Z 437.727,A -85,B 0,C 180,E1 -6372.876,E2 -6372.876} C_VEL
LIN {X 0,Y 491.893,Z 451.327,A -85,B 0,C 180,E1 -6373.396,E2 -6373.396} C_VEL
LIN {X 0,Y 491.446,Z 463.7,A -85,B 0,C 180,E1 -6374.021,E2 -6374.021} C_VEL
LIN {X 0,Y 490.866,Z 476.634,A -85,B 0,C 180,E1 -6374.853,E2 -6374.853} C_VEL
LIN {X 0,Y 490.301,Z 488.355,A -85,B 0,C 180,E1 -6375.791,E2 -6375.791} C_VEL
LIN {X 0,Y 489.728,Z 499.176,A -85,B 0,C 180,E1 -6376.842,E2 -6376.842} C_VEL
LIN {X 0,Y 489.292,Z 509.42,A -85,B 0,C 180,E1 -6378.049,E2 -6378.049} C_VEL
LIN {X 0,Y 488.874,Z 517.767,A -85,B 0,C 180,E1 -6379.229,E2 -6379.229} C_VEL
LIN {X 0,Y 488.503,Z 526.279,A -85,B 0,C 180,E1 -6380.686,E2 -6380.686} C_VEL
LIN {X 0,Y 488.225,Z 533.136,A -85,B 0,C 180,E1 -6382.14,E2 -6382.14} C_VEL
LIN {X 0,Y 488.06,Z 539.155,A -85,B 0,C 180,E1 -6383.762,E2 -6383.762} C_VEL
LIN {X 0,Y 487.964,Z 542.777,A -85,B 0,C 180,E1 -6385.043,E2 -6385.043} C_VEL
LIN {X 0,Y 487.962,Z 546.193,A -85,B 0,C 180,E1 -6386.697,E2 -6386.697} C_VEL
LIN {X 0,Y 487.89,Z 548.225,A -85,B 0,C 180,E1 -6388.349,E2 -6388.349} C_VEL
LIN {X 0,Y 487.818,Z 548.927,A -85,B 0,C 180,E1 -6390,E2 -6390} C_VEL
LIN {X 0,Y 487.888,Z 548.306,A -85,B 0,C 180,E1 -6391.651,E2 -6391.651} C_VEL
LIN {X 0,Y 487.961,Z 546.347,A -85,B 0,C 180,E1 -6393.303,E2 -6393.303} C_VEL
LIN {X 0,Y 487.964,Z 543.005,A -85,B 0,C 180,E1 -6394.957,E2 -6394.957} C_VEL
LIN {X 0,Y 488.14,Z 538.181,A -85,B 0,C 180,E1 -6396.614,E2 -6396.614} C_VEL
LIN {X 0,Y 488.295,Z 531.723,A -85,B 0,C 180,E1 -6398.275,E2 -6398.275} C_VEL
LIN {X 0,Y 488.612,Z 524.531,A -85,B 0,C 180,E1 -6399.73,E2 -6399.73} C_VEL
LIN {X 0,Y 488.937,Z 516.997,A -85,B 0,C 180,E1 -6400.979,E2 -6400.979} C_VEL
LIN {X 0,Y 489.289,Z 507.983,A -85,B 0,C 180,E1 -6402.227,E2 -6402.227} C_VEL
LIN {X 0,Y 489.743,Z 498.938,A -85,B 0,C 180,E1 -6403.274,E2 -6403.274} C_VEL
LIN {X 0,Y 490.309,Z 488.184,A -85,B 0,C 180,E1 -6404.315,E2 -6404.315} C_VEL
LIN {X 0,Y 490.848,Z 476.419,A -85,B 0,C 180,E1 -6405.253,E2 -6405.253} C_VEL
LIN {X 0,Y 491.461,Z 463.436,A -85,B 0,C 180,E1 -6406.085,E2 -6406.085} C_VEL
LIN {X 0,Y 491.902,Z 450.537,A -85,B 0,C 180,E1 -6406.732,E2 -6406.732} C_VEL
LIN {X 0,Y 492.303,Z 436.766,A -85,B 0,C 180,E1 -6407.245,E2 -6407.245} C_VEL
LIN {X 0,Y 492.601,Z 422.79,A -85,B 0,C 180,E1 -6407.594,E2 -6407.594} C_VEL
LIN {X 0,Y 493.548,Z 303.312,A -85,B 0,C 180,E1 -6409.371,E2 -6409.371} C_VEL
LIN {X 0,Y 490.36,Z 287.169,A -85,B 0,C 180,E1 -6409.77,E2 -6409.77} C_VEL
LIN {X 0,Y 490.856,Z 274.655,A -85,B 0,C 180,E1 -6411.855,E2 -6411.855} C_VEL
LIN {X 0,Y 491.029,Z 268.484,A -85,B 0,C 180,E1 -6412.923,E2 -6412.923} C_VEL
LIN {X 0,Y 488.752,Z 257.363,A -85,B 0,C 180,E1 -6415.054,E2 -6415.054} C_VEL
LIN {X 0,Y 488.746,Z 257.221,A -85,B 0,C 180,E1 -6417.396,E2 -6417.396} C_VEL
LIN {X 0,Y 488.709,Z 257.233,A -85,B 0,C 180,E1 -6420.362,E2 -6420.362} C_VEL
LIN {X 0,Y 488.734,Z 257.232,A -85,B 0,C 180,E1 -6423.484,E2 -6423.484} C_VEL
LIN {X 0,Y 488.685,Z 257.235,A -85,B 0,C 180,E1 -6426.355,E2 -6426.355} C_VEL
LIN {X 0,Y 488.698,Z 257.234,A -85,B 0,C 180,E1 -6429.253,E2 -6429.253} C_VEL
LIN {X 0,Y 488.72,Z 257.226,A -85,B 0,C 180,E1 -6431.601,E2 -6431.601} C_VEL
LIN {X 0,Y 488.708,Z 257.231,A -85,B 0,C 180,E1 -6434.801,E2 -6434.801} C_VEL
LIN {X 0,Y 488.687,Z 257.226,A -85,B 0,C 180,E1 -6437.474,E2 -6437.474} C_VEL
LIN {X 0,Y 488.728,Z 257.227,A -85,B 0,C 180,E1 -6439.676,E2 -6439.676} C_VEL
LIN {X 0,Y 488.674,Z 257.236,A -85,B 0,C 180,E1 -6442.277,E2 -6442.277} C_VEL
LIN {X 0,Y 488.723,Z 257.225,A -85,B 0,C 180,E1 -6445.051,E2 -6445.051} C_VEL
LIN {X 0,Y 488.699,Z 257.222,A -85,B 0,C 180,E1 -6448.045,E2 -6448.045} C_VEL
LIN {X 0,Y 488.727,Z 257.231,A -85,B 0,C 180,E1 -6450.73,E2 -6450.73} C_VEL
LIN {X 0,Y 488.749,Z 257.222,A -85,B 0,C 180,E1 -6453.527,E2 -6453.527} C_VEL
LIN {X 0,Y 488.684,Z 257.234,A -85,B 0,C 180,E1 -6456.254,E2 -6456.254} C_VEL
LIN {X 0,Y 488.738,Z 257.226,A -85,B 0,C 180,E1 -6459.175,E2 -6459.175} C_VEL
LIN {X 0,Y 488.727,Z 257.231,A -85,B 0,C 180,E1 -6462.423,E2 -6462.423} C_VEL
LIN {X 0,Y 488.753,Z 257.224,A -85,B 0,C 180,E1 -6464.999,E2 -6464.999} C_VEL
LIN {X 0,Y 488.799,Z 257.222,A -85,B 0,C 180,E1 -6468.387,E2 -6468.387} C_VEL
LIN {X 0,Y 488.809,Z 257.212,A -85,B 0,C 180,E1 -6471.733,E2 -6471.733} C_VEL
LIN {X 0,Y 488.853,Z 257.215,A -85,B 0,C 180,E1 -6474.224,E2 -6474.224} C_VEL
LIN {X 0,Y 488.953,Z 257.191,A -85,B 0,C 180,E1 -6477.529,E2 -6477.529} C_VEL
LIN {X 0,Y 488.959,Z 257.199,A -85,B 0,C 180,E1 -6480,E2 -6480} C_VEL
LIN {X 0,Y 488.953,Z 257.203,A -85,B 0,C 180,E1 -6482.471,E2 -6482.471} C_VEL
LIN {X 0,Y 488.847,Z 257.211,A -85,B 0,C 180,E1 -6485.776,E2 -6485.776} C_VEL
LIN {X 0,Y 488.809,Z 257.224,A -85,B 0,C 180,E1 -6488.266,E2 -6488.266} C_VEL
LIN {X 0,Y 488.796,Z 257.216,A -85,B 0,C 180,E1 -6491.613,E2 -6491.613} C_VEL
LIN {X 0,Y 488.753,Z 257.222,A -85,B 0,C 180,E1 -6495.001,E2 -6495.001} C_VEL
LIN {X 0,Y 488.746,Z 257.231,A -85,B 0,C 180,E1 -6498.442,E2 -6498.442} C_VEL
LIN {X 0,Y 488.698,Z 257.229,A -85,B 0,C 180,E1 -6501.071,E2 -6501.071} C_VEL
LIN {X 0,Y 488.685,Z 257.234,A -85,B 0,C 180,E1 -6503.746,E2 -6503.746} C_VEL
LIN {X 0,Y 488.784,Z 257.216,A -85,B 0,C 180,E1 -6506.944,E2 -6506.944} C_VEL
LIN {X 0,Y 488.727,Z 257.232,A -85,B 0,C 180,E1 -6510.219,E2 -6510.219} C_VEL
LIN {X 0,Y 488.729,Z 257.22,A -85,B 0,C 180,E1 -6513.485,E2 -6513.485} C_VEL
LIN {X 0,Y 488.683,Z 257.232,A -85,B 0,C 180,E1 -6516.356,E2 -6516.356} C_VEL
LIN {X 0,Y 488.696,Z 257.234,A -85,B 0,C 180,E1 -6519.255,E2 -6519.255} C_VEL
LIN {X 0,Y 488.703,Z 257.234,A -85,B 0,C 180,E1 -6521.601,E2 -6521.601} C_VEL
LIN {X 0,Y 488.707,Z 257.23,A -85,B 0,C 180,E1 -6524.802,E2 -6524.802} C_VEL
LIN {X 0,Y 488.731,Z 257.227,A -85,B 0,C 180,E1 -6527.48,E2 -6527.48} C_VEL
LIN {X 0,Y 488.739,Z 257.228,A -85,B 0,C 180,E1 -6530.75,E2 -6530.75} C_VEL
LIN {X 0,Y 488.674,Z 257.24,A -85,B 0,C 180,E1 -6533.869,E2 -6533.869} C_VEL
LIN {X 0,Y 488.736,Z 257.225,A -85,B 0,C 180,E1 -6536.878,E2 -6536.878} C_VEL
LIN {X 0,Y 488.722,Z 257.214,A -85,B 0,C 180,E1 -6539.781,E2 -6539.781} C_VEL
LIN {X 0,Y 488.791,Z 257.215,A -85,B 0,C 180,E1 -6543.057,E2 -6543.057} C_VEL
LIN {X 0,Y 488.807,Z 257.384,A -85,B 0,C 180,E1 -6543.876,E2 -6543.876} C_VEL
LIN {X 0,Y 491.178,Z 268.91,A -85,B 0,C 180,E1 -6545.979,E2 -6545.979} C_VEL
LIN {X 0,Y 491.183,Z 274.024,A -85,B 0,C 180,E1 -6546.829,E2 -6546.829} C_VEL
LIN {X 0,Y 490.393,Z 291.5,A -85,B 0,C 180,E1 -6549.664,E2 -6549.664} C_VEL
LIN {X 0,Y 490.33,Z 295.553,A -85,B 0,C 180,E1 -6550.272,E2 -6550.272} C_VEL
LIN {X 0,Y 493.531,Z 313.615,A -85,B 0,C 180,E1 -6550.697,E2 -6550.697} C_VEL
LIN {X 0,Y 492.531,Z 433.321,A -85,B 0,C 180,E1 -6552.483,E2 -6552.483} C_VEL
LIN {X 0,Y 492.129,Z 447.805,A -85,B 0,C 180,E1 -6552.87,E2 -6552.87} C_VEL
LIN {X 0,Y 491.726,Z 462.269,A -85,B 0,C 180,E1 -6553.444,E2 -6553.444} C_VEL
LIN {X 0,Y 491.267,Z 475.08,A -85,B 0,C 180,E1 -6554.122,E2 -6554.122} C_VEL
LIN {X 0,Y 490.632,Z 487.55,A -85,B 0,C 180,E1 -6554.952,E2 -6554.952} C_VEL
LIN {X 0,Y 490.129,Z 498.945,A -85,B 0,C 180,E1 -6555.892,E2 -6555.892} C_VEL
LIN {X 0,Y 489.572,Z 509.415,A -85,B 0,C 180,E1 -6556.933,E2 -6556.933} C_VEL
LIN {X 0,Y 489.166,Z 520.119,A -85,B 0,C 180,E1 -6558.224,E2 -6558.224} C_VEL
LIN {X 0,Y 488.667,Z 529.687,A -85,B 0,C 180,E1 -6559.644,E2 -6559.644} C_VEL
LIN {X 0,Y 488.35,Z 537.656,A -85,B 0,C 180,E1 -6561.1,E2 -6561.1} C_VEL
LIN {X 0,Y 488.108,Z 544.071,A -85,B 0,C 180,E1 -6562.555,E2 -6562.555} C_VEL
LIN {X 0,Y 488.018,Z 548.511,A -85,B 0,C 180,E1 -6563.799,E2 -6563.799} C_VEL
LIN {X 0,Y 487.961,Z 552.006,A -85,B 0,C 180,E1 -6565.043,E2 -6565.043} C_VEL
LIN {X 0,Y 487.955,Z 555.404,A -85,B 0,C 180,E1 -6566.697,E2 -6566.697} C_VEL
LIN {X 0,Y 487.886,Z 557.413,A -85,B 0,C 180,E1 -6568.349,E2 -6568.349} C_VEL
LIN {X 0,Y 487.817,Z 558.079,A -85,B 0,C 180,E1 -6570,E2 -6570} C_VEL
LIN {X 0,Y 487.886,Z 557.414,A -85,B 0,C 180,E1 -6571.651,E2 -6571.651} C_VEL
LIN {X 0,Y 487.955,Z 555.408,A -85,B 0,C 180,E1 -6573.303,E2 -6573.303} C_VEL
LIN {X 0,Y 487.961,Z 552.009,A -85,B 0,C 180,E1 -6574.957,E2 -6574.957} C_VEL
LIN {X 0,Y 488.045,Z 547.601,A -85,B 0,C 180,E1 -6576.475,E2 -6576.475} C_VEL
LIN {X 0,Y 488.168,Z 542.401,A -85,B 0,C 180,E1 -6577.861,E2 -6577.861} C_VEL
LIN {X 0,Y 488.429,Z 535.559,A -85,B 0,C 180,E1 -6579.316,E2 -6579.316} C_VEL
LIN {X 0,Y 488.806,Z 527.063,A -85,B 0,C 180,E1 -6580.772,E2 -6580.772} C_VEL
LIN {X 0,Y 489.171,Z 518.81,A -85,B 0,C 180,E1 -6581.945,E2 -6581.945} C_VEL
LIN {X 0,Y 489.599,Z 509.413,A -85,B 0,C 180,E1 -6583.066,E2 -6583.066} C_VEL
LIN {X 0,Y 490.109,Z 498.941,A -85,B 0,C 180,E1 -6584.109,E2 -6584.109} C_VEL
LIN {X 0,Y 490.646,Z 487.548,A -85,B 0,C 180,E1 -6585.047,E2 -6585.047} C_VEL
LIN {X 0,Y 491.249,Z 475.073,A -85,B 0,C 180,E1 -6585.879,E2 -6585.879} C_VEL
LIN {X 0,Y 491.752,Z 462.249,A -85,B 0,C 180,E1 -6586.555,E2 -6586.555} C_VEL
LIN {X 0,Y 492.164,Z 447.759,A -85,B 0,C 180,E1 -6587.129,E2 -6587.129} C_VEL
LIN {X 0,Y 492.525,Z 433.294,A -85,B 0,C 180,E1 -6587.517,E2 -6587.517} C_VEL
LIN {X 0,Y 493.529,Z 313.081,A -85,B 0,C 180,E1 -6589.311,E2 -6589.311} C_VEL
LIN {X 0,Y 490.303,Z 295.432,A -85,B 0,C 180,E1 -6589.735,E2 -6589.735} C_VEL
LIN {X 0,Y 490.917,Z 279.394,A -85,B 0,C 180,E1 -6592.295,E2 -6592.295} C_VEL
LIN {X 0,Y 491.32,Z 270.628,A -85,B 0,C 180,E1 -6593.726,E2 -6593.726} C_VEL
LIN {X 0,Y 490.134,Z 263.691,A -85,B 0,C 180,E1 -6594.947,E2 -6594.947} C_VEL
LIN {X 0,Y 488.807,Z 257.376,A -85,B 0,C 180,E1 -6596.124,E2 -6596.124} C_VEL
LIN {X 0,Y 488.722,Z 257.213,A -85,B 0,C 180,E1 -6599.27,E2 -6599.27} C_VEL
LIN {X 0,Y 488.702,Z 257.235,A -85,B 0,C 180,E1 -6602.146,E2 -6602.146} C_VEL
LIN {X 0,Y 488.715,Z 257.233,A -85,B 0,C 180,E1 -6605.114,E2 -6605.114} C_VEL
LIN {X 0,Y 488.676,Z 257.235,A -85,B 0,C 180,E1 -6608.199,E2 -6608.199} C_VEL
LIN {X 0,Y 488.715,Z 257.231,A -85,B 0,C 180,E1 -6610.344,E2 -6610.344} C_VEL
LIN {X 0,Y 488.733,Z 257.229,A -85,B 0,C 180,E1 -6612.829,E2 -6612.829} C_VEL
LIN {X 0,Y 488.695,Z 257.235,A -85,B 0,C 180,E1 -6615.976,E2 -6615.976} C_VEL
LIN {X 0,Y 488.703,Z 257.232,A -85,B 0,C 180,E1 -6618.584,E2 -6618.584} C_VEL
LIN {X 0,Y 488.699,Z 257.232,A -85,B 0,C 180,E1 -6620.947,E2 -6620.947} C_VEL
LIN {X 0,Y 488.68,Z 257.231,A -85,B 0,C 180,E1 -6623.868,E2 -6623.868} C_VEL
LIN {X 0,Y 488.733,Z 257.219,A -85,B 0,C 180,E1 -6626.877,E2 -6626.877} C_VEL
LIN {X 0,Y 488.728,Z 257.232,A -85,B 0,C 180,E1 -6629.781,E2 -6629.781} C_VEL
LIN {X 0,Y 488.792,Z 257.216,A -85,B 0,C 180,E1 -6633.054,E2 -6633.054} C_VEL
LIN {X 0,Y 488.686,Z 257.234,A -85,B 0,C 180,E1 -6636.254,E2 -6636.254} C_VEL
LIN {X 0,Y 488.738,Z 257.225,A -85,B 0,C 180,E1 -6639.175,E2 -6639.175} C_VEL
LIN {X 0,Y 488.727,Z 257.225,A -85,B 0,C 180,E1 -6642.423,E2 -6642.423} C_VEL
LIN {X 0,Y 488.754,Z 257.222,A -85,B 0,C 180,E1 -6644.999,E2 -6644.999} C_VEL
LIN {X 0,Y 488.797,Z 257.216,A -85,B 0,C 180,E1 -6648.387,E2 -6648.387} C_VEL
LIN {X 0,Y 488.809,Z 257.224,A -85,B 0,C 180,E1 -6651.734,E2 -6651.734} C_VEL
LIN {X 0,Y 488.847,Z 257.211,A -85,B 0,C 180,E1 -6654.224,E2 -6654.224} C_VEL
LIN {X 0,Y 488.953,Z 257.202,A -85,B 0,C 180,E1 -6657.529,E2 -6657.529} C_VEL
LIN {X 0,Y 488.947,Z 257.2,A -85,B 0,C 180,E1 -6660.824,E2 -6660.824} C_VEL
LIN {X 0,Y 488.953,Z 257.191,A -85,B 0,C 180,E1 -6662.471,E2 -6662.471} C_VEL
LIN {X 0,Y 488.853,Z 257.215,A -85,B 0,C 180,E1 -6665.776,E2 -6665.776} C_VEL
LIN {X 0,Y 488.809,Z 257.212,A -85,B 0,C 180,E1 -6668.267,E2 -6668.267} C_VEL
LIN {X 0,Y 488.797,Z 257.223,A -85,B 0,C 180,E1 -6671.613,E2 -6671.613} C_VEL
LIN {X 0,Y 488.754,Z 257.224,A -85,B 0,C 180,E1 -6675.001,E2 -6675.001} C_VEL
LIN {X 0,Y 488.747,Z 257.226,A -85,B 0,C 180,E1 -6678.443,E2 -6678.443} C_VEL
LIN {X 0,Y 488.699,Z 257.232,A -85,B 0,C 180,E1 -6681.071,E2 -6681.071} C_VEL
LIN {X 0,Y 488.685,Z 257.234,A -85,B 0,C 180,E1 -6683.746,E2 -6683.746} C_VEL
LIN {X 0,Y 488.785,Z 257.222,A -85,B 0,C 180,E1 -6686.944,E2 -6686.944} C_VEL
LIN {X 0,Y 488.728,Z 257.227,A -85,B 0,C 180,E1 -6690.219,E2 -6690.219} C_VEL
LIN {X 0,Y 488.73,Z 257.211,A -85,B 0,C 180,E1 -6693.485,E2 -6693.485} C_VEL
LIN {X 0,Y 488.684,Z 257.232,A -85,B 0,C 180,E1 -6696.356,E2 -6696.356} C_VEL
LIN {X 0,Y 488.733,Z 257.225,A -85,B 0,C 180,E1 -6699.251,E2 -6699.251} C_VEL
LIN {X 0,Y 488.707,Z 257.216,A -85,B 0,C 180,E1 -6701.601,E2 -6701.601} C_VEL
LIN {X 0,Y 488.708,Z 257.237,A -85,B 0,C 180,E1 -6704.802,E2 -6704.802} C_VEL
LIN {X 0,Y 488.692,Z 257.222,A -85,B 0,C 180,E1 -6707.476,E2 -6707.476} C_VEL
LIN {X 0,Y 488.73,Z 257.228,A -85,B 0,C 180,E1 -6709.677,E2 -6709.677} C_VEL
LIN {X 0,Y 488.68,Z 257.236,A -85,B 0,C 180,E1 -6712.842,E2 -6712.842} C_VEL
LIN {X 0,Y 488.733,Z 257.227,A -85,B 0,C 180,E1 -6715.888,E2 -6715.888} C_VEL
LIN {X 0,Y 488.692,Z 257.235,A -85,B 0,C 180,E1 -6718.821,E2 -6718.821} C_VEL
LIN {X 0,Y 488.745,Z 257.218,A -85,B 0,C 180,E1 -6721.672,E2 -6721.672} C_VEL
LIN {X 0,Y 488.725,Z 257.225,A -85,B 0,C 180,E1 -6724.353,E2 -6724.353} C_VEL
LIN {X 0,Y 488.536,Z 257.78,A -85,B 0,C 180,E1 -6724.807,E2 -6724.807} C_VEL
LIN {X 0,Y 488.045,Z 259.18,A -85,B 0,C 180,E1 -6725.236,E2 -6725.236} C_VEL
LIN {X 0,Y 486.557,Z 263.363,A -85,B 0,C 180,E1 -6726.029,E2 -6726.029} C_VEL
LIN {X 0,Y 484.984,Z 268.076,A -85,B 0,C 180,E1 -6726.785,E2 -6726.785} C_VEL
LIN {X 0,Y 484.115,Z 272.687,A -85,B 0,C 180,E1 -6727.558,E2 -6727.558} C_VEL
LIN {X 0,Y 483.466,Z 287.103,A -85,B 0,C 180,E1 -6730.02,E2 -6730.02} C_VEL
LIN {X 0,Y 486.83,Z 303.928,A -85,B 0,C 180,E1 -6730.451,E2 -6730.451} C_VEL
LIN {X 0,Y 485.832,Z 423.763,A -85,B 0,C 180,E1 -6732.261,E2 -6732.261} C_VEL
LIN {X 0,Y 485.48,Z 437.567,A -85,B 0,C 180,E1 -6732.621,E2 -6732.621} C_VEL
LIN {X 0,Y 485.089,Z 451.404,A -85,B 0,C 180,E1 -6733.157,E2 -6733.157} C_VEL
LIN {X 0,Y 484.613,Z 463.775,A -85,B 0,C 180,E1 -6733.79,E2 -6733.79} C_VEL
LIN {X 0,Y 484.021,Z 476.707,A -85,B 0,C 180,E1 -6734.634,E2 -6734.634} C_VEL
LIN {X 0,Y 483.412,Z 488.428,A -85,B 0,C 180,E1 -6735.584,E2 -6735.584} C_VEL
LIN {X 0,Y 482.728,Z 500.124,A -85,B 0,C 180,E1 -6736.744,E2 -6736.744} C_VEL
LIN {X 0,Y 482.302,Z 509.736,A -85,B 0,C 180,E1 -6737.906,E2 -6737.906} C_VEL
LIN {X 0,Y 481.79,Z 519.188,A -85,B 0,C 180,E1 -6739.281,E2 -6739.281} C_VEL
LIN {X 0,Y 481.409,Z 527.451,A -85,B 0,C 180,E1 -6740.759,E2 -6740.759} C_VEL
LIN {X 0,Y 481.172,Z 533.206,A -85,B 0,C 180,E1 -6742.024,E2 -6742.024} C_VEL
LIN {X 0,Y 481.034,Z 538.525,A -85,B 0,C 180,E1 -6743.461,E2 -6743.461} C_VEL
LIN {X 0,Y 480.9,Z 542.845,A -85,B 0,C 180,E1 -6744.97,E2 -6744.97} C_VEL
LIN {X 0,Y 480.887,Z 546.261,A -85,B 0,C 180,E1 -6746.649,E2 -6746.649} C_VEL
LIN {X 0,Y 480.791,Z 548.292,A -85,B 0,C 180,E1 -6748.325,E2 -6748.325} C_VEL
LIN {X 0,Y 480.742,Z 548.994,A -85,B 0,C 180,E1 -6750,E2 -6750} C_VEL
LIN {X 0,Y 480.79,Z 548.372,A -85,B 0,C 180,E1 -6751.675,E2 -6751.675} C_VEL
LIN {X 0,Y 480.887,Z 546.412,A -85,B 0,C 180,E1 -6753.351,E2 -6753.351} C_VEL
LIN {X 0,Y 480.899,Z 543.07,A -85,B 0,C 180,E1 -6755.03,E2 -6755.03} C_VEL
LIN {X 0,Y 481.054,Z 538.246,A -85,B 0,C 180,E1 -6756.712,E2 -6756.712} C_VEL
LIN {X 0,Y 481.247,Z 531.787,A -85,B 0,C 180,E1 -6758.397,E2 -6758.397} C_VEL
LIN {X 0,Y 481.575,Z 524.596,A -85,B 0,C 180,E1 -6759.873,E2 -6759.873} C_VEL
LIN {X 0,Y 481.949,Z 517.061,A -85,B 0,C 180,E1 -6761.14,E2 -6761.14} C_VEL
LIN {X 0,Y 482.29,Z 508.62,A -85,B 0,C 180,E1 -6762.332,E2 -6762.332} C_VEL
LIN {X 0,Y 482.818,Z 499,A -85,B 0,C 180,E1 -6763.467,E2 -6763.467} C_VEL
LIN {X 0,Y 483.404,Z 488.245,A -85,B 0,C 180,E1 -6764.524,E2 -6764.524} C_VEL
LIN {X 0,Y 483.989,Z 476.479,A -85,B 0,C 180,E1 -6765.475,E2 -6765.475} C_VEL
LIN {X 0,Y 484.633,Z 463.495,A -85,B 0,C 180,E1 -6766.318,E2 -6766.318} C_VEL
LIN {X 0,Y 485.155,Z 449.902,A -85,B 0,C 180,E1 -6767.003,E2 -6767.003} C_VEL
LIN {X 0,Y 485.543,Z 436.414,A -85,B 0,C 180,E1 -6767.505,E2 -6767.505} C_VEL
LIN {X 0,Y 485.836,Z 422.83,A -85,B 0,C 180,E1 -6767.848,E2 -6767.848} C_VEL
LIN {X 0,Y 486.887,Z 304.426,A -85,B 0,C 180,E1 -6769.63,E2 -6769.63} C_VEL
LIN {X 0,Y 483.48,Z 287.259,A -85,B 0,C 180,E1 -6770.061,E2 -6770.061} C_VEL
LIN {X 0,Y 483.822,Z 277.963,A -85,B 0,C 180,E1 -6771.617,E2 -6771.617} C_VEL
LIN {X 0,Y 484.173,Z 270.893,A -85,B 0,C 180,E1 -6772.847,E2 -6772.847} C_VEL
LIN {X 0,Y 482.233,Z 260.755,A -85,B 0,C 180,E1 -6774.771,E2 -6774.771} C_VEL
LIN {X 0,Y 481.693,Z 258.137,A -85,B 0,C 180,E1 -6775.346,E2 -6775.346} C_VEL
LIN {X 0,Y 481.7,Z 258.094,A -85,B 0,C 180,E1 -6777.831,E2 -6777.831} C_VEL
LIN {X 0,Y 481.645,Z 258.113,A -85,B 0,C 180,E1 -6780.71,E2 -6780.71} C_VEL
LIN {X 0,Y 481.695,Z 258.106,A -85,B 0,C 180,E1 -6783.732,E2 -6783.732} C_VEL
LIN {X 0,Y 481.626,Z 258.115,A -85,B 0,C 180,E1 -6786.746,E2 -6786.746} C_VEL
LIN {X 0,Y 481.674,Z 258.11,A -85,B 0,C 180,E1 -6789.94,E2 -6789.94} C_VEL
LIN {X 0,Y 481.662,Z 258.104,A -85,B 0,C 180,E1 -6793.296,E2 -6793.296} C_VEL
LIN {X 0,Y 481.654,Z 258.113,A -85,B 0,C 180,E1 -6795.64,E2 -6795.64} C_VEL
LIN {X 0,Y 481.663,Z 258.096,A -85,B 0,C 180,E1 -6798.959,E2 -6798.959} C_VEL
LIN {X 0,Y 481.692,Z 258.107,A -85,B 0,C 180,E1 -6801.143,E2 -6801.143} C_VEL
LIN {X 0,Y 481.662,Z 258.109,A -85,B 0,C 180,E1 -6804.794,E2 -6804.794} C_VEL
LIN {X 0,Y 481.667,Z 258.095,A -85,B 0,C 180,E1 -6807.325,E2 -6807.325} C_VEL
LIN {X 0,Y 481.681,Z 258.105,A -85,B 0,C 180,E1 -6810.259,E2 -6810.259} C_VEL
LIN {X 0,Y 481.738,Z 258.1,A -85,B 0,C 180,E1 -6813.111,E2 -6813.111} C_VEL
LIN {X 0,Y 481.669,Z 258.107,A -85,B 0,C 180,E1 -6815.886,E2 -6815.886} C_VEL
LIN {X 0,Y 481.694,Z 258.104,A -85,B 0,C 180,E1 -6819.027,E2 -6819.027} C_VEL
LIN {X 0,Y 481.699,Z 258.104,A -85,B 0,C 180,E1 -6822.158,E2 -6822.158} C_VEL
LIN {X 0,Y 481.734,Z 258.099,A -85,B 0,C 180,E1 -6824.775,E2 -6824.775} C_VEL
LIN {X 0,Y 481.744,Z 258.099,A -85,B 0,C 180,E1 -6828.215,E2 -6828.215} C_VEL
LIN {X 0,Y 481.754,Z 258.09,A -85,B 0,C 180,E1 -6831.611,E2 -6831.611} C_VEL
LIN {X 0,Y 481.813,Z 258.091,A -85,B 0,C 180,E1 -6834.139,E2 -6834.139} C_VEL
LIN {X 0,Y 481.92,Z 258.067,A -85,B 0,C 180,E1 -6837.492,E2 -6837.492} C_VEL
LIN {X 0,Y 481.931,Z 258.075,A -85,B 0,C 180,E1 -6840,E2 -6840} C_VEL
LIN {X 0,Y 481.92,Z 258.078,A -85,B 0,C 180,E1 -6842.507,E2 -6842.507} C_VEL
LIN {X 0,Y 481.808,Z 258.088,A -85,B 0,C 180,E1 -6845.86,E2 -6845.86} C_VEL
LIN {X 0,Y 481.755,Z 258.101,A -85,B 0,C 180,E1 -6848.388,E2 -6848.388} C_VEL
LIN {X 0,Y 481.741,Z 258.096,A -85,B 0,C 180,E1 -6851.785,E2 -6851.785} C_VEL
LIN {X 0,Y 481.733,Z 258.096,A -85,B 0,C 180,E1 -6855.224,E2 -6855.224} C_VEL
LIN {X 0,Y 481.703,Z 258.105,A -85,B 0,C 180,E1 -6858.722,E2 -6858.722} C_VEL
LIN {X 0,Y 481.638,Z 258.109,A -85,B 0,C 180,E1 -6861.395,E2 -6861.395} C_VEL
LIN {X 0,Y 481.669,Z 258.113,A -85,B 0,C 180,E1 -6864.114,E2 -6864.114} C_VEL
LIN {X 0,Y 481.739,Z 258.094,A -85,B 0,C 180,E1 -6867.14,E2 -6867.14} C_VEL
LIN {X 0,Y 481.681,Z 258.11,A -85,B 0,C 180,E1 -6869.741,E2 -6869.741} C_VEL
LIN {X 0,Y 481.666,Z 258.098,A -85,B 0,C 180,E1 -6872.675,E2 -6872.675} C_VEL
LIN {X 0,Y 481.636,Z 258.1,A -85,B 0,C 180,E1 -6875.71,E2 -6875.71} C_VEL
LIN {X 0,Y 481.665,Z 258.108,A -85,B 0,C 180,E1 -6878.86,E2 -6878.86} C_VEL
LIN {X 0,Y 481.648,Z 258.116,A -85,B 0,C 180,E1 -6881.914,E2 -6881.914} C_VEL
LIN {X 0,Y 481.654,Z 258.109,A -85,B 0,C 180,E1 -6884.458,E2 -6884.458} C_VEL
LIN {X 0,Y 481.685,Z 258.105,A -85,B 0,C 180,E1 -6886.846,E2 -6886.846} C_VEL
LIN {X 0,Y 481.685,Z 258.109,A -85,B 0,C 180,E1 -6890.062,E2 -6890.062} C_VEL
LIN {X 0,Y 481.622,Z 258.11,A -85,B 0,C 180,E1 -6893.254,E2 -6893.254} C_VEL
LIN {X 0,Y 481.707,Z 258.099,A -85,B 0,C 180,E1 -6896.331,E2 -6896.331} C_VEL
LIN {X 0,Y 481.648,Z 258.098,A -85,B 0,C 180,E1 -6899.418,E2 -6899.418} C_VEL
LIN {X 0,Y 481.699,Z 258.109,A -85,B 0,C 180,E1 -6902.169,E2 -6902.169} C_VEL
LIN {X 0,Y 481.761,Z 258.157,A -85,B 0,C 180,E1 -6903.581,E2 -6903.581} C_VEL
LIN {X 0,Y 482.254,Z 260.493,A -85,B 0,C 180,E1 -6904.075,E2 -6904.075} C_VEL
LIN {X 0,Y 484.388,Z 271.532,A -85,B 0,C 180,E1 -6906.074,E2 -6906.074} C_VEL
LIN {X 0,Y 483.662,Z 288.751,A -85,B 0,C 180,E1 -6908.923,E2 -6908.923} C_VEL
LIN {X 0,Y 483.388,Z 295.147,A -85,B 0,C 180,E1 -6909.95,E2 -6909.95} C_VEL
LIN {X 0,Y 484.253,Z 299.724,A -85,B 0,C 180,E1 -6910.099,E2 -6910.099} C_VEL
LIN {X 0,Y 486.824,Z 314.613,A -85,B 0,C 180,E1 -6910.436,E2 -6910.436} C_VEL
LIN {X 0,Y 485.775,Z 432.021,A -85,B 0,C 180,E1 -6912.205,E2 -6912.205} C_VEL
LIN {X 0,Y 485.419,Z 446.148,A -85,B 0,C 180,E1 -6912.569,E2 -6912.569} C_VEL
LIN {X 0,Y 484.977,Z 460.06,A -85,B 0,C 180,E1 -6913.104,E2 -6913.104} C_VEL
LIN {X 0,Y 484.463,Z 473.25,A -85,B 0,C 180,E1 -6913.785,E2 -6913.785} C_VEL
LIN {X 0,Y 483.846,Z 486.059,A -85,B 0,C 180,E1 -6914.628,E2 -6914.628} C_VEL
LIN {X 0,Y 483.264,Z 497.705,A -85,B 0,C 180,E1 -6915.579,E2 -6915.579} C_VEL
LIN {X 0,Y 482.732,Z 507.396,A -85,B 0,C 180,E1 -6916.53,E2 -6916.53} C_VEL
LIN {X 0,Y 482.25,Z 517.281,A -85,B 0,C 180,E1 -6917.689,E2 -6917.689} C_VEL
LIN {X 0,Y 481.788,Z 526.998,A -85,B 0,C 180,E1 -6919.069,E2 -6919.069} C_VEL
LIN {X 0,Y 481.388,Z 535.492,A -85,B 0,C 180,E1 -6920.547,E2 -6920.547} C_VEL
LIN {X 0,Y 481.119,Z 542.336,A -85,B 0,C 180,E1 -6922.023,E2 -6922.023} C_VEL
LIN {X 0,Y 480.965,Z 547.886,A -85,B 0,C 180,E1 -6923.533,E2 -6923.533} C_VEL
LIN {X 0,Y 480.895,Z 551.94,A -85,B 0,C 180,E1 -6924.97,E2 -6924.97} C_VEL
LIN {X 0,Y 480.861,Z 555.337,A -85,B 0,C 180,E1 -6926.649,E2 -6926.649} C_VEL
LIN {X 0,Y 480.787,Z 557.346,A -85,B 0,C 180,E1 -6928.325,E2 -6928.325} C_VEL
LIN {X 0,Y 480.741,Z 558.012,A -85,B 0,C 180,E1 -6930,E2 -6930} C_VEL
LIN {X 0,Y 480.787,Z 557.348,A -85,B 0,C 180,E1 -6931.675,E2 -6931.675} C_VEL
LIN {X 0,Y 480.861,Z 555.341,A -85,B 0,C 180,E1 -6933.352,E2 -6933.352} C_VEL
LIN {X 0,Y 480.895,Z 551.943,A -85,B 0,C 180,E1 -6935.03,E2 -6935.03} C_VEL
LIN {X 0,Y 480.962,Z 547.051,A -85,B 0,C 180,E1 -6936.713,E2 -6936.713} C_VEL
LIN {X 0,Y 481.203,Z 540.522,A -85,B 0,C 180,E1 -6938.398,E2 -6938.398} C_VEL
LIN {X 0,Y 481.467,Z 533.255,A -85,B 0,C 180,E1 -6939.876,E2 -6939.876} C_VEL
LIN {X 0,Y 481.93,Z 524.256,A -85,B 0,C 180,E1 -6941.354,E2 -6941.354} C_VEL
LIN {X 0,Y 482.365,Z 514.81,A -85,B 0,C 180,E1 -6942.624,E2 -6942.624} C_VEL
LIN {X 0,Y 482.902,Z 504.352,A -85,B 0,C 180,E1 -6943.787,E2 -6943.787} C_VEL
LIN {X 0,Y 483.486,Z 492.812,A -85,B 0,C 180,E1 -6944.844,E2 -6944.844} C_VEL
LIN {X 0,Y 484.186,Z 480.009,A -85,B 0,C 180,E1 -6945.792,E2 -6945.792} C_VEL
LIN {X 0,Y 484.7,Z 467.503,A -85,B 0,C 180,E1 -6946.532,E2 -6946.532} C_VEL
LIN {X 0,Y 485.191,Z 454.37,A -85,B 0,C 180,E1 -6947.132,E2 -6947.132} C_VEL
LIN {X 0,Y 485.597,Z 440.147,A -85,B 0,C 180,E1 -6947.604,E2 -6947.604} C_VEL
LIN {X 0,Y 485.871,Z 425.934,A -85,B 0,C 180,E1 -6947.901,E2 -6947.901} C_VEL
LIN {X 0,Y 486.85,Z 313.921,A -85,B 0,C 180,E1 -6949.572,E2 -6949.572} C_VEL
LIN {X 0,Y 483.384,Z 295.506,A -85,B 0,C 180,E1 -6950.02,E2 -6950.02} C_VEL
LIN {X 0,Y 483.657,Z 288.738,A -85,B 0,C 180,E1 -6951.078,E2 -6951.078} C_VEL
LIN {X 0,Y 484.448,Z 272.378,A -85,B 0,C 180,E1 -6953.779,E2 -6953.779} C_VEL
LIN {X 0,Y 482.913,Z 263.688,A -85,B 0,C 180,E1 -6955.336,E2 -6955.336} C_VEL
LIN {X 0,Y 481.791,Z 258.497,A -85,B 0,C 180,E1 -6956.3,E2 -6956.3} C_VEL
LIN {X 0,Y 481.728,Z 258.089,A -85,B 0,C 180,E1 -6956.538,E2 -6956.538} C_VEL
LIN {X 0,Y 481.677,Z 258.088,A -85,B 0,C 180,E1 -6959.741,E2 -6959.741} C_VEL
LIN {X 0,Y 481.67,Z 258.11,A -85,B 0,C 180,E1 -6962.674,E2 -6962.674} C_VEL
LIN {X 0,Y 481.634,Z 258.114,A -85,B 0,C 180,E1 -6965.709,E2 -6965.709} C_VEL
LIN {X 0,Y 481.667,Z 258.112,A -85,B 0,C 180,E1 -6968.859,E2 -6968.859} C_VEL
LIN {X 0,Y 481.662,Z 258.102,A -85,B 0,C 180,E1 -6972.158,E2 -6972.158} C_VEL
LIN {X 0,Y 481.655,Z 258.109,A -85,B 0,C 180,E1 -6975.542,E2 -6975.542} C_VEL
LIN {X 0,Y 481.652,Z 258.107,A -85,B 0,C 180,E1 -6978.958,E2 -6978.958} C_VEL
LIN {X 0,Y 481.651,Z 258.115,A -85,B 0,C 180,E1 -6981.992,E2 -6981.992} C_VEL
LIN {X 0,Y 481.687,Z 258.087,A -85,B 0,C 180,E1 -6985.318,E2 -6985.318} C_VEL
LIN {X 0,Y 481.642,Z 258.115,A -85,B 0,C 180,E1 -6988.311,E2 -6988.311} C_VEL
LIN {X 0,Y 481.7,Z 258.103,A -85,B 0,C 180,E1 -6991.219,E2 -6991.219} C_VEL
LIN {X 0,Y 481.699,Z 258.109,A -85,B 0,C 180,E1 -6994.043,E2 -6994.043} C_VEL
LIN {X 0,Y 481.667,Z 258.104,A -85,B 0,C 180,E1 -6996.811,E2 -6996.811} C_VEL
LIN {X 0,Y 481.688,Z 258.105,A -85,B 0,C 180,E1 -6999.502,E2 -6999.502} C_VEL
LIN {X 0,Y 481.699,Z 258.103,A -85,B 0,C 180,E1 -7002.158,E2 -7002.158} C_VEL
LIN {X 0,Y 481.734,Z 258.096,A -85,B 0,C 180,E1 -7004.776,E2 -7004.776} C_VEL
LIN {X 0,Y 481.742,Z 258.096,A -85,B 0,C 180,E1 -7008.215,E2 -7008.215} C_VEL
LIN {X 0,Y 481.755,Z 258.1,A -85,B 0,C 180,E1 -7011.612,E2 -7011.612} C_VEL
LIN {X 0,Y 481.808,Z 258.088,A -85,B 0,C 180,E1 -7014.14,E2 -7014.14} C_VEL
LIN {X 0,Y 481.92,Z 258.077,A -85,B 0,C 180,E1 -7017.493,E2 -7017.493} C_VEL
LIN {X 0,Y 481.898,Z 258.078,A -85,B 0,C 180,E1 -7020.836,E2 -7020.836} C_VEL
LIN {X 0,Y 481.92,Z 258.067,A -85,B 0,C 180,E1 -7022.508,E2 -7022.508} C_VEL
LIN {X 0,Y 481.813,Z 258.091,A -85,B 0,C 180,E1 -7025.861,E2 -7025.861} C_VEL
LIN {X 0,Y 481.755,Z 258.09,A -85,B 0,C 180,E1 -7028.389,E2 -7028.389} C_VEL
LIN {X 0,Y 481.742,Z 258.1,A -85,B 0,C 180,E1 -7031.785,E2 -7031.785} C_VEL
LIN {X 0,Y 481.734,Z 258.098,A -85,B 0,C 180,E1 -7035.225,E2 -7035.225} C_VEL
LIN {X 0,Y 481.704,Z 258.106,A -85,B 0,C 180,E1 -7038.722,E2 -7038.722} C_VEL
LIN {X 0,Y 481.638,Z 258.113,A -85,B 0,C 180,E1 -7041.395,E2 -7041.395} C_VEL
LIN {X 0,Y 481.669,Z 258.107,A -85,B 0,C 180,E1 -7044.114,E2 -7044.114} C_VEL
LIN {X 0,Y 481.74,Z 258.102,A -85,B 0,C 180,E1 -7047.14,E2 -7047.14} C_VEL
LIN {X 0,Y 481.682,Z 258.105,A -85,B 0,C 180,E1 -7049.741,E2 -7049.741} C_VEL
LIN {X 0,Y 481.667,Z 258.095,A -85,B 0,C 180,E1 -7052.675,E2 -7052.675} C_VEL
LIN {X 0,Y 481.637,Z 258.107,A -85,B 0,C 180,E1 -7055.71,E2 -7055.71} C_VEL
LIN {X 0,Y 481.706,Z 258.1,A -85,B 0,C 180,E1 -7059.354,E2 -7059.354} C_VEL
LIN {X 0,Y 481.645,Z 258.097,A -85,B 0,C 180,E1 -7062.161,E2 -7062.161} C_VEL
LIN {X 0,Y 481.657,Z 258.109,A -85,B 0,C 180,E1 -7065.544,E2 -7065.544} C_VEL
LIN {X 0,Y 481.66,Z 258.099,A -85,B 0,C 180,E1 -7068.087,E2 -7068.087} C_VEL
LIN {X 0,Y 481.669,Z 258.106,A -85,B 0,C 180,E1 -7071.142,E2 -7071.142} C_VEL
LIN {X 0,Y 481.666,Z 258.11,A -85,B 0,C 180,E1 -7074.796,E2 -7074.796} C_VEL
LIN {X 0,Y 481.671,Z 258.109,A -85,B 0,C 180,E1 -7077.327,E2 -7077.327} C_VEL
LIN {X 0,Y 481.679,Z 258.112,A -85,B 0,C 180,E1 -7080.26,E2 -7080.26} C_VEL
LIN {X 0,Y 481.746,Z 258.099,A -85,B 0,C 180,E1 -7083.113,E2 -7083.113} C_VEL
LIN {X 0,Y 481.694,Z 258.175,A -85,B 0,C 180,E1 -7084.769,E2 -7084.769} C_VEL
LIN {X 0,Y 482.658,Z 262.775,A -85,B 0,C 180,E1 -7085.711,E2 -7085.711} C_VEL
LIN {X 0,Y 484.156,Z 270.382,A -85,B 0,C 180,E1 -7087.152,E2 -7087.152} C_VEL
LIN {X 0,Y 484.115,Z 272.687,A -85,B 0,C 180,E1 -7087.558,E2 -7087.558} C_VEL
LIN {X 0,Y 483.345,Z 275.006,A -85,B 0,C 180,E1 -7087.929,E2 -7087.929} C_VEL
LIN {X 0,Y 480.386,Z 278.93,A -85,B 0,C 180,E1 -7088.478,E2 -7088.478} C_VEL
LIN {X 0,Y 477.408,Z 282.864,A -85,B 0,C 180,E1 -7089.032,E2 -7089.032} C_VEL
LIN {X 0,Y 476.626,Z 285.2,A -85,B 0,C 180,E1 -7089.409,E2 -7089.409} C_VEL
LIN {X 0,Y 476.607,Z 287.496,A -85,B 0,C 180,E1 -7089.741,E2 -7089.741} C_VEL
LIN {X 0,Y 480.117,Z 304.82,A -85,B 0,C 180,E1 -7090.178,E2 -7090.178} C_VEL
LIN {X 0,Y 479.1,Z 422.397,A -85,B 0,C 180,E1 -7091.976,E2 -7091.976} C_VEL
LIN {X 0,Y 478.791,Z 436.066,A -85,B 0,C 180,E1 -7092.32,E2 -7092.32} C_VEL
LIN {X 0,Y 478.378,Z 449.346,A -85,B 0,C 180,E1 -7092.814,E2 -7092.814} C_VEL
LIN {X 0,Y 477.857,Z 462.009,A -85,B 0,C 180,E1 -7093.444,E2 -7093.444} C_VEL
LIN {X 0,Y 477.228,Z 475.356,A -85,B 0,C 180,E1 -7094.3,E2 -7094.3} C_VEL
LIN {X 0,Y 476.584,Z 487.328,A -85,B 0,C 180,E1 -7095.263,E2 -7095.263} C_VEL
LIN {X 0,Y 475.924,Z 498.247,A -85,B 0,C 180,E1 -7096.334,E2 -7096.334} C_VEL
LIN {X 0,Y 475.303,Z 508.533,A -85,B 0,C 180,E1 -7097.555,E2 -7097.555} C_VEL
LIN {X 0,Y 475.005,Z 516.556,A -85,B 0,C 180,E1 -7098.695,E2 -7098.695} C_VEL
LIN {X 0,Y 474.517,Z 525.305,A -85,B 0,C 180,E1 -7100.193,E2 -7100.193} C_VEL
LIN {X 0,Y 474.231,Z 531.47,A -85,B 0,C 180,E1 -7101.478,E2 -7101.478} C_VEL
LIN {X 0,Y 473.96,Z 538.009,A -85,B 0,C 180,E1 -7103.187,E2 -7103.187} C_VEL
LIN {X 0,Y 473.838,Z 542.913,A -85,B 0,C 180,E1 -7104.894,E2 -7104.894} C_VEL
LIN {X 0,Y 473.796,Z 546.328,A -85,B 0,C 180,E1 -7106.598,E2 -7106.598} C_VEL
LIN {X 0,Y 473.697,Z 548.359,A -85,B 0,C 180,E1 -7108.3,E2 -7108.3} C_VEL
LIN {X 0,Y 473.668,Z 549.06,A -85,B 0,C 180,E1 -7110,E2 -7110} C_VEL
LIN {X 0,Y 473.696,Z 548.438,A -85,B 0,C 180,E1 -7111.7,E2 -7111.7} C_VEL
LIN {X 0,Y 473.795,Z 546.478,A -85,B 0,C 180,E1 -7113.401,E2 -7113.401} C_VEL
LIN {X 0,Y 473.838,Z 543.135,A -85,B 0,C 180,E1 -7115.105,E2 -7115.105} C_VEL
LIN {X 0,Y 473.976,Z 538.311,A -85,B 0,C 180,E1 -7116.812,E2 -7116.812} C_VEL
LIN {X 0,Y 474.21,Z 531.852,A -85,B 0,C 180,E1 -7118.523,E2 -7118.523} C_VEL
LIN {X 0,Y 474.538,Z 524.66,A -85,B 0,C 180,E1 -7120.021,E2 -7120.021} C_VEL
LIN {X 0,Y 475.012,Z 515.766,A -85,B 0,C 180,E1 -7121.521,E2 -7121.521} C_VEL
LIN {X 0,Y 475.499,Z 506.422,A -85,B 0,C 180,E1 -7122.809,E2 -7122.809} C_VEL
LIN {X 0,Y 476.047,Z 496.073,A -85,B 0,C 180,E1 -7123.989,E2 -7123.989} C_VEL
LIN {X 0,Y 476.705,Z 484.654,A -85,B 0,C 180,E1 -7125.06,E2 -7125.06} C_VEL
LIN {X 0,Y 477.406,Z 471.997,A -85,B 0,C 180,E1 -7126.023,E2 -7126.023} C_VEL
LIN {X 0,Y 477.954,Z 459.888,A -85,B 0,C 180,E1 -7126.761,E2 -7126.761} C_VEL
LIN {X 0,Y 478.492,Z 446.071,A -85,B 0,C 180,E1 -7127.413,E2 -7127.413} C_VEL
LIN {X 0,Y 478.879,Z 431.885,A -85,B 0,C 180,E1 -7127.895,E2 -7127.895} C_VEL
LIN {X 0,Y 479.143,Z 418.358,A -85,B 0,C 180,E1 -7128.188,E2 -7128.188} C_VEL
LIN {X 0,Y 480.199,Z 305.539,A -85,B 0,C 180,E1 -7129.899,E2 -7129.899} C_VEL
LIN {X 0,Y 476.604,Z 287.455,A -85,B 0,C 180,E1 -7130.357,E2 -7130.357} C_VEL
LIN {X 0,Y 476.678,Z 284.963,A -85,B 0,C 180,E1 -7130.722,E2 -7130.722} C_VEL
LIN {X 0,Y 477.263,Z 272.225,A -85,B 0,C 180,E1 -7132.968,E2 -7132.968} C_VEL
LIN {X 0,Y 475.021,Z 260.813,A -85,B 0,C 180,E1 -7135.173,E2 -7135.173} C_VEL
LIN {X 0,Y 474.674,Z 259.03,A -85,B 0,C 180,E1 -7135.585,E2 -7135.585} C_VEL
LIN {X 0,Y 474.646,Z 258.971,A -85,B 0,C 180,E1 -7138.282,E2 -7138.282} C_VEL
LIN {X 0,Y 474.598,Z 258.99,A -85,B 0,C 180,E1 -7141.217,E2 -7141.217} C_VEL
LIN {X 0,Y 474.632,Z 258.983,A -85,B 0,C 180,E1 -7144.24,E2 -7144.24} C_VEL
LIN {X 0,Y 474.589,Z 258.99,A -85,B 0,C 180,E1 -7147.383,E2 -7147.383} C_VEL
LIN {X 0,Y 474.625,Z 258.992,A -85,B 0,C 180,E1 -7149.647,E2 -7149.647} C_VEL
LIN {X 0,Y 474.632,Z 258.975,A -85,B 0,C 180,E1 -7152.931,E2 -7152.931} C_VEL
LIN {X 0,Y 474.605,Z 258.988,A -85,B 0,C 180,E1 -7155.894,E2 -7155.894} C_VEL
LIN {X 0,Y 474.636,Z 258.971,A -85,B 0,C 180,E1 -7159.038,E2 -7159.038} C_VEL
LIN {X 0,Y 474.611,Z 258.991,A -85,B 0,C 180,E1 -7161.702,E2 -7161.702} C_VEL
LIN {X 0,Y 474.624,Z 258.985,A -85,B 0,C 180,E1 -7164.725,E2 -7164.725} C_VEL
LIN {X 0,Y 474.631,Z 258.975,A -85,B 0,C 180,E1 -7167.787,E2 -7167.787} C_VEL
LIN {X 0,Y 474.626,Z 258.99,A -85,B 0,C 180,E1 -7170.882,E2 -7170.882} C_VEL
LIN {X 0,Y 474.653,Z 258.977,A -85,B 0,C 180,E1 -7173.628,E2 -7173.628} C_VEL
LIN {X 0,Y 474.628,Z 258.988,A -85,B 0,C 180,E1 -7176.641,E2 -7176.641} C_VEL
LIN {X 0,Y 474.646,Z 258.978,A -85,B 0,C 180,E1 -7180.089,E2 -7180.089} C_VEL
LIN {X 0,Y 474.643,Z 258.99,A -85,B 0,C 180,E1 -7182.774,E2 -7182.774} C_VEL
LIN {X 0,Y 474.64,Z 258.979,A -85,B 0,C 180,E1 -7185.421,E2 -7185.421} C_VEL
LIN {X 0,Y 474.697,Z 258.976,A -85,B 0,C 180,E1 -7188.037,E2 -7188.037} C_VEL
LIN {X 0,Y 474.72,Z 258.966,A -85,B 0,C 180,E1 -7191.486,E2 -7191.486} C_VEL
LIN {X 0,Y 474.775,Z 258.967,A -85,B 0,C 180,E1 -7194.052,E2 -7194.052} C_VEL
LIN {X 0,Y 474.886,Z 258.943,A -85,B 0,C 180,E1 -7197.455,E2 -7197.455} C_VEL
LIN {X 0,Y 474.868,Z 258.958,A -85,B 0,C 180,E1 -7200.848,E2 -7200.848} C_VEL
LIN {X 0,Y 474.886,Z 258.953,A -85,B 0,C 180,E1 -7202.545,E2 -7202.545} C_VEL
LIN {X 0,Y 474.771,Z 258.966,A -85,B 0,C 180,E1 -7205.948,E2 -7205.948} C_VEL
LIN {X 0,Y 474.72,Z 258.975,A -85,B 0,C 180,E1 -7208.514,E2 -7208.514} C_VEL
LIN {X 0,Y 474.695,Z 258.975,A -85,B 0,C 180,E1 -7211.963,E2 -7211.963} C_VEL
LIN {X 0,Y 474.691,Z 258.974,A -85,B 0,C 180,E1 -7215.456,E2 -7215.456} C_VEL
LIN {X 0,Y 474.656,Z 258.981,A -85,B 0,C 180,E1 -7219.011,E2 -7219.011} C_VEL
LIN {X 0,Y 474.582,Z 258.99,A -85,B 0,C 180,E1 -7221.729,E2 -7221.729} C_VEL
LIN {X 0,Y 474.651,Z 258.985,A -85,B 0,C 180,E1 -7224.493,E2 -7224.493} C_VEL
LIN {X 0,Y 474.691,Z 258.972,A -85,B 0,C 180,E1 -7227.339,E2 -7227.339} C_VEL
LIN {X 0,Y 474.603,Z 258.987,A -85,B 0,C 180,E1 -7230.812,E2 -7230.812} C_VEL
LIN {X 0,Y 474.631,Z 258.967,A -85,B 0,C 180,E1 -7233.985,E2 -7233.985} C_VEL
LIN {X 0,Y 474.569,Z 258.988,A -85,B 0,C 180,E1 -7236.9,E2 -7236.9} C_VEL
LIN {X 0,Y 474.622,Z 258.99,A -85,B 0,C 180,E1 -7239.648,E2 -7239.648} C_VEL
LIN {X 0,Y 474.609,Z 258.988,A -85,B 0,C 180,E1 -7242.935,E2 -7242.935} C_VEL
LIN {X 0,Y 474.614,Z 258.99,A -85,B 0,C 180,E1 -7245.897,E2 -7245.897} C_VEL
LIN {X 0,Y 474.641,Z 258.975,A -85,B 0,C 180,E1 -7249.039,E2 -7249.039} C_VEL
LIN {X 0,Y 474.612,Z 258.987,A -85,B 0,C 180,E1 -7251.704,E2 -7251.704} C_VEL
LIN {X 0,Y 474.621,Z 258.988,A -85,B 0,C 180,E1 -7254.726,E2 -7254.726} C_VEL
LIN {X 0,Y 474.634,Z 258.989,A -85,B 0,C 180,E1 -7257.788,E2 -7257.788} C_VEL
LIN {X 0,Y 474.622,Z 258.969,A -85,B 0,C 180,E1 -7260.885,E2 -7260.885} C_VEL
LIN {X 0,Y 474.723,Z 259.066,A -85,B 0,C 180,E1 -7263.337,E2 -7263.337} C_VEL
LIN {X 0,Y 475.55,Z 262.827,A -85,B 0,C 180,E1 -7264.101,E2 -7264.101} C_VEL
LIN {X 0,Y 477.523,Z 273.314,A -85,B 0,C 180,E1 -7266.023,E2 -7266.023} C_VEL
LIN {X 0,Y 476.715,Z 290.031,A -85,B 0,C 180,E1 -7268.827,E2 -7268.827} C_VEL
LIN {X 0,Y 476.5,Z 295.084,A -85,B 0,C 180,E1 -7269.647,E2 -7269.647} C_VEL
LIN {X 0,Y 477.346,Z 299.532,A -85,B 0,C 180,E1 -7269.796,E2 -7269.796} C_VEL
LIN {X 0,Y 480.079,Z 314.436,A -85,B 0,C 180,E1 -7270.148,E2 -7270.148} C_VEL
LIN {X 0,Y 479.186,Z 420.593,A -85,B 0,C 180,E1 -7271.758,E2 -7271.758} C_VEL
LIN {X 0,Y 478.917,Z 436.627,A -85,B 0,C 180,E1 -7272.051,E2 -7272.051} C_VEL
LIN {X 0,Y 478.512,Z 450.753,A -85,B 0,C 180,E1 -7272.478,E2 -7272.478} C_VEL
LIN {X 0,Y 478.017,Z 464.672,A -85,B 0,C 180,E1 -7273.078,E2 -7273.078} C_VEL
LIN {X 0,Y 477.468,Z 476.719,A -85,B 0,C 180,E1 -7273.76,E2 -7273.76} C_VEL
LIN {X 0,Y 476.816,Z 488.847,A -85,B 0,C 180,E1 -7274.615,E2 -7274.615} C_VEL
LIN {X 0,Y 476.174,Z 501.083,A -85,B 0,C 180,E1 -7275.687,E2 -7275.687} C_VEL
LIN {X 0,Y 475.583,Z 511.181,A -85,B 0,C 180,E1 -7276.759,E2 -7276.759} C_VEL
LIN {X 0,Y 475.082,Z 521.219,A -85,B 0,C 180,E1 -7278.048,E2 -7278.048} C_VEL
LIN {X 0,Y 474.61,Z 529.555,A -85,B 0,C 180,E1 -7279.333,E2 -7279.333} C_VEL
LIN {X 0,Y 474.255,Z 537.523,A -85,B 0,C 180,E1 -7280.834,E2 -7280.834} C_VEL
LIN {X 0,Y 473.973,Z 543.938,A -85,B 0,C 180,E1 -7282.331,E2 -7282.331} C_VEL
LIN {X 0,Y 473.834,Z 549.625,A -85,B 0,C 180,E1 -7284.041,E2 -7284.041} C_VEL
LIN {X 0,Y 473.827,Z 551.874,A -85,B 0,C 180,E1 -7284.894,E2 -7284.894} C_VEL
LIN {X 0,Y 473.755,Z 555.271,A -85,B 0,C 180,E1 -7286.598,E2 -7286.598} C_VEL
LIN {X 0,Y 473.692,Z 557.28,A -85,B 0,C 180,E1 -7288.3,E2 -7288.3} C_VEL
LIN {X 0,Y 473.668,Z 557.946,A -85,B 0,C 180,E1 -7290,E2 -7290} C_VEL
LIN {X 0,Y 473.692,Z 557.281,A -85,B 0,C 180,E1 -7291.7,E2 -7291.7} C_VEL
LIN {X 0,Y 473.755,Z 555.274,A -85,B 0,C 180,E1 -7293.402,E2 -7293.402} C_VEL
LIN {X 0,Y 473.829,Z 551.876,A -85,B 0,C 180,E1 -7295.106,E2 -7295.106} C_VEL
LIN {X 0,Y 473.892,Z 546.983,A -85,B 0,C 180,E1 -7296.814,E2 -7296.814} C_VEL
LIN {X 0,Y 474.131,Z 540.454,A -85,B 0,C 180,E1 -7298.524,E2 -7298.524} C_VEL
LIN {X 0,Y 474.431,Z 533.187,A -85,B 0,C 180,E1 -7300.024,E2 -7300.024} C_VEL
LIN {X 0,Y 474.94,Z 524.188,A -85,B 0,C 180,E1 -7301.523,E2 -7301.523} C_VEL
LIN {X 0,Y 475.4,Z 514.742,A -85,B 0,C 180,E1 -7302.812,E2 -7302.812} C_VEL
LIN {X 0,Y 475.97,Z 504.283,A -85,B 0,C 180,E1 -7303.992,E2 -7303.992} C_VEL
LIN {X 0,Y 476.596,Z 492.743,A -85,B 0,C 180,E1 -7305.064,E2 -7305.064} C_VEL
LIN {X 0,Y 477.338,Z 479.939,A -85,B 0,C 180,E1 -7306.025,E2 -7306.025} C_VEL
LIN {X 0,Y 477.871,Z 467.818,A -85,B 0,C 180,E1 -7306.754,E2 -7306.754} C_VEL
LIN {X 0,Y 478.415,Z 454.299,A -85,B 0,C 180,E1 -7307.383,E2 -7307.383} C_VEL
LIN {X 0,Y 478.836,Z 440.073,A -85,B 0,C 180,E1 -7307.861,E2 -7307.861} C_VEL
LIN {X 0,Y 479.117,Z 425.854,A -85,B 0,C 180,E1 -7308.162,E2 -7308.162} C_VEL
LIN {X 0,Y 480.134,Z 314.699,A -85,B 0,C 180,E1 -7309.844,E2 -7309.844} C_VEL
LIN {X 0,Y 476.514,Z 295.25,A -85,B 0,C 180,E1 -7310.335,E2 -7310.335} C_VEL
LIN {X 0,Y 477.447,Z 276.582,A -85,B 0,C 180,E1 -7313.418,E2 -7313.418} C_VEL
LIN {X 0,Y 477.426,Z 272.48,A -85,B 0,C 180,E1 -7314.122,E2 -7314.122} C_VEL
LIN {X 0,Y 474.82,Z 259.734,A -85,B 0,C 180,E1 -7316.48,E2 -7316.48} C_VEL
LIN {X 0,Y 474.734,Z 258.988,A -85,B 0,C 180,E1 -7316.722,E2 -7316.722} C_VEL
LIN {X 0,Y 474.603,Z 258.971,A -85,B 0,C 180,E1 -7320.23,E2 -7320.23} C_VEL
LIN {X 0,Y 474.641,Z 258.979,A -85,B 0,C 180,E1 -7323.219,E2 -7323.219} C_VEL
LIN {X 0,Y 474.586,Z 258.991,A -85,B 0,C 180,E1 -7326.323,E2 -7326.323} C_VEL
LIN {X 0,Y 474.624,Z 258.987,A -85,B 0,C 180,E1 -7329.647,E2 -7329.647} C_VEL
LIN {X 0,Y 474.64,Z 258.984,A -85,B 0,C 180,E1 -7332.93,E2 -7332.93} C_VEL
LIN {X 0,Y 474.605,Z 258.989,A -85,B 0,C 180,E1 -7335.895,E2 -7335.895} C_VEL
LIN {X 0,Y 474.623,Z 258.982,A -85,B 0,C 180,E1 -7339.04,E2 -7339.04} C_VEL
LIN {X 0,Y 474.605,Z 258.99,A -85,B 0,C 180,E1 -7341.703,E2 -7341.703} C_VEL
LIN {X 0,Y 474.624,Z 258.967,A -85,B 0,C 180,E1 -7344.726,E2 -7344.726} C_VEL
LIN {X 0,Y 474.631,Z 258.978,A -85,B 0,C 180,E1 -7347.787,E2 -7347.787} C_VEL
LIN {X 0,Y 474.625,Z 258.984,A -85,B 0,C 180,E1 -7350.882,E2 -7350.882} C_VEL
LIN {X 0,Y 474.659,Z 258.979,A -85,B 0,C 180,E1 -7353.628,E2 -7353.628} C_VEL
LIN {X 0,Y 474.628,Z 258.981,A -85,B 0,C 180,E1 -7356.641,E2 -7356.641} C_VEL
LIN {X 0,Y 474.647,Z 258.987,A -85,B 0,C 180,E1 -7360.089,E2 -7360.089} C_VEL
LIN {X 0,Y 474.643,Z 258.977,A -85,B 0,C 180,E1 -7362.774,E2 -7362.774} C_VEL
LIN {X 0,Y 474.64,Z 258.984,A -85,B 0,C 180,E1 -7365.421,E2 -7365.421} C_VEL
LIN {X 0,Y 474.695,Z 258.975,A -85,B 0,C 180,E1 -7368.037,E2 -7368.037} C_VEL
LIN {X 0,Y 474.72,Z 258.974,A -85,B 0,C 180,E1 -7371.486,E2 -7371.486} C_VEL
LIN {X 0,Y 474.771,Z 258.966,A -85,B 0,C 180,E1 -7374.052,E2 -7374.052} C_VEL
LIN {X 0,Y 474.886,Z 258.952,A -85,B 0,C 180,E1 -7377.455,E2 -7377.455} C_VEL
LIN {X 0,Y 474.903,Z 258.951,A -85,B 0,C 180,E1 -7380,E2 -7380} C_VEL
LIN {X 0,Y 474.887,Z 258.942,A -85,B 0,C 180,E1 -7382.545,E2 -7382.545} C_VEL
LIN {X 0,Y 474.775,Z 258.967,A -85,B 0,C 180,E1 -7385.948,E2 -7385.948} C_VEL
LIN {X 0,Y 474.72,Z 258.966,A -85,B 0,C 180,E1 -7388.514,E2 -7388.514} C_VEL
LIN {X 0,Y 474.696,Z 258.977,A -85,B 0,C 180,E1 -7391.963,E2 -7391.963} C_VEL
LIN {X 0,Y 474.692,Z 258.976,A -85,B 0,C 180,E1 -7395.456,E2 -7395.456} C_VEL
LIN {X 0,Y 474.657,Z 258.987,A -85,B 0,C 180,E1 -7399.011,E2 -7399.011} C_VEL
LIN {X 0,Y 474.581,Z 258.989,A -85,B 0,C 180,E1 -7401.729,E2 -7401.729} C_VEL
LIN {X 0,Y 474.652,Z 258.983,A -85,B 0,C 180,E1 -7404.493,E2 -7404.493} C_VEL
LIN {X 0,Y 474.693,Z 258.98,A -85,B 0,C 180,E1 -7407.339,E2 -7407.339} C_VEL
LIN {X 0,Y 474.605,Z 258.988,A -85,B 0,C 180,E1 -7410.812,E2 -7410.812} C_VEL
LIN {X 0,Y 474.633,Z 258.964,A -85,B 0,C 180,E1 -7413.985,E2 -7413.985} C_VEL
LIN {X 0,Y 474.571,Z 258.997,A -85,B 0,C 180,E1 -7416.901,E2 -7416.901} C_VEL
LIN {X 0,Y 474.643,Z 258.978,A -85,B 0,C 180,E1 -7419.651,E2 -7419.651} C_VEL
LIN {X 0,Y 474.628,Z 258.981,A -85,B 0,C 180,E1 -7422.933,E2 -7422.933} C_VEL
LIN {X 0,Y 474.612,Z 258.987,A -85,B 0,C 180,E1 -7425.897,E2 -7425.897} C_VEL
LIN {X 0,Y 474.63,Z 258.988,A -85,B 0,C 180,E1 -7429.041,E2 -7429.041} C_VEL
LIN {X 0,Y 474.608,Z 258.984,A -85,B 0,C 180,E1 -7431.705,E2 -7431.705} C_VEL
LIN {X 0,Y 474.627,Z 258.987,A -85,B 0,C 180,E1 -7434.727,E2 -7434.727} C_VEL
LIN {X 0,Y 474.635,Z 258.987,A -85,B 0,C 180,E1 -7437.788,E2 -7437.788} C_VEL
LIN {X 0,Y 474.624,Z 258.981,A -85,B 0,C 180,E1 -7440.885,E2 -7440.885} C_VEL
LIN {X 0,Y 474.655,Z 258.987,A -85,B 0,C 180,E1 -7443.629,E2 -7443.629} C_VEL
LIN {X 0,Y 474.689,Z 259.175,A -85,B 0,C 180,E1 -7444.574,E2 -7444.574} C_VEL
LIN {X 0,Y 477.228,Z 271.718,A -85,B 0,C 180,E1 -7447.03,E2 -7447.03} C_VEL
LIN {X 0,Y 476.626,Z 285.2,A -85,B 0,C 180,E1 -7449.409,E2 -7449.409} C_VEL
LIN {X 0,Y 475.938,Z 286.75,A -85,B 0,C 180,E1 -7449.565,E2 -7449.565} C_VEL
